// TIA Portal V18 export
FUNCTION_BLOCK "V90_Servo"   // FB2500, LAD
{ S7_Optimized_Access := 'TRUE' }
// stored: AutoNumber false, MemoryReserve 100, SetENOAutomatically false
   VAR
      Servo_380A1 { S7_SetPoint := 'True'} : "fbV90Ctrl";   // *
      Servo_381A1 { S7_SetPoint := 'True'} : "fbV90Ctrl";   // *
      Servo_382A1 { S7_SetPoint := 'True'} : "fbV90Ctrl";   // *
      Servo_383A1 { S7_SetPoint := 'True'} : "fbV90Ctrl";   // *
      Servo1 { S7_SetPoint := 'True'} : "SevroStart&PosCheck";
      Servo2 { S7_SetPoint := 'True'} : "SevroStart&PosCheck";
      Servo3 { S7_SetPoint := 'True'} : "SevroStart&PosCheck";
      Servo4 { S7_SetPoint := 'True'} : "SevroStart&PosCheck";
      Servo2SafetyPos { S7_SetPoint := 'True'} : DInt;
      Servo4SafetyPos { S7_SetPoint := 'True'} : DInt;
      IEC_Timer_0_Instance { S7_SetPoint := 'True'} : TON_TIME;
      P { S7_SetPoint := 'True'} : Array[0..10] of Bool;
      MC_MOVEJOG_Instance { S7_SetPoint := 'True'} : MC_MOVEJOG;
      MC_POWER_Instance { S7_SetPoint := 'True'} : MC_POWER;
      BasicPosControl { S7_SetPoint := 'True'} : BasicPosControl;
   END_VAR
   VAR_TEMP
      Sevro1ActPos : Real;
      Sevro1StartList : Bool;
      Sevro2ActPos : Real;
      Sevro2StartList : Bool;
      Sevro3ActPos : Real;
      Sevro3StartList : Bool;
      Sevro4ActPos : Real;
      Sevro4StartList : Bool;
      dummy : Bool;
      gotopos : Real;
      speed : Int;
   END_VAR
   VAR_TEMP   // added for the SCL form of the ladder/FBD networks
      _w1 : Bool;
      _w2 : Bool;
      _w3 : Bool;
      _w4 : Bool;
      _w5 : Bool;
   END_VAR
BEGIN

REGION Network 1: <<<<<<<<<<<<<<<<<<<<<380A1 Servo>>>>>>>>>>>>>>>>>>>>>>>>>
END_REGION

REGION Network 2: negtive motion/action/...automaticly
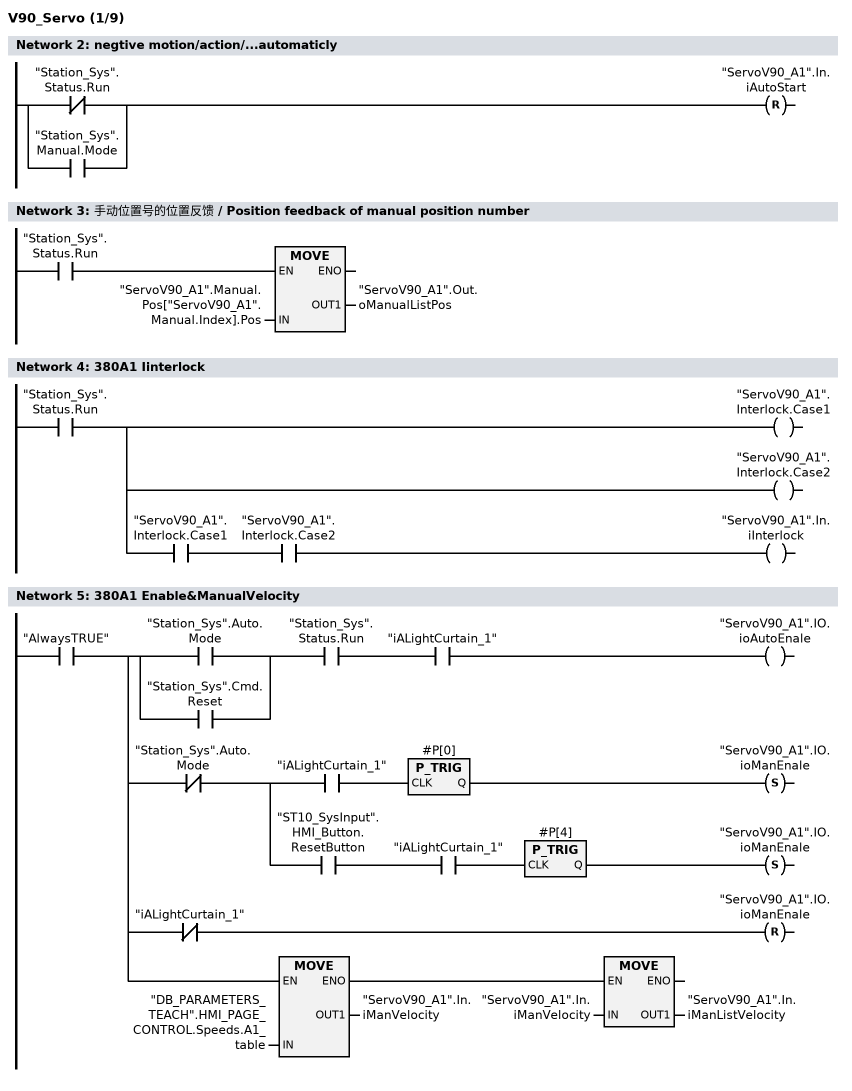
   RUNG wire#powerrail
      I_Contact( "Station_Sys".Status.Run )
      wire#w1
      R_Coil( "ServoV90_A1".In.iAutoStart )
   END_RUNG
   RUNG wire#powerrail
      Contact( "Station_Sys".Manual.Mode )
   END_RUNG wire#w1
   // the same network as SCL:
   IF NOT "Station_Sys".Status.Run OR "Station_Sys".Manual.Mode THEN
       "ServoV90_A1".In.iAutoStart := FALSE;
   END_IF;
END_REGION

REGION Network 3: 手动位置号的位置反馈 / Position feedback of manual position number
   RUNG wire#powerrail
      Contact( "Station_Sys".Status.Run )
      Move(in := "ServoV90_A1".Manual.Pos["ServoV90_A1".Manual.Index].Pos, out1 => "ServoV90_A1".Out.oManualListPos)
   END_RUNG
   // the same network as SCL:
   IF "Station_Sys".Status.Run THEN
       "ServoV90_A1".Out.oManualListPos := "ServoV90_A1".Manual.Pos["ServoV90_A1".Manual.Index].Pos;
   END_IF;
END_REGION

REGION Network 4: 380A1 Iinterlock
   RUNG wire#powerrail
      Contact( "Station_Sys".Status.Run )
      wire#w1
      Coil( "ServoV90_A1".Interlock.Case1 )
   END_RUNG
   RUNG wire#w1
      Coil( "ServoV90_A1".Interlock.Case2 )
   END_RUNG
   RUNG wire#w1
      Contact( "ServoV90_A1".Interlock.Case1 )
      Contact( "ServoV90_A1".Interlock.Case2 )
      Coil( "ServoV90_A1".In.iInterlock )
   END_RUNG
   // the same network as SCL:
   "ServoV90_A1".Interlock.Case1 := "Station_Sys".Status.Run;
   "ServoV90_A1".Interlock.Case2 := "Station_Sys".Status.Run;
   "ServoV90_A1".In.iInterlock := "Station_Sys".Status.Run AND "ServoV90_A1".Interlock.Case1 AND "ServoV90_A1".Interlock.Case2;
END_REGION

REGION Network 5: 380A1 Enable&ManualVelocity
   RUNG wire#powerrail
      Contact( "AlwaysTRUE" )
      wire#w1
      Contact( "Station_Sys".Auto.Mode )
      wire#w2
      Contact( "Station_Sys".Status.Run )
      Contact( "iALightCurtain_1" )
      Coil( "ServoV90_A1".IO.ioAutoEnale )
   END_RUNG
   RUNG wire#w1
      Contact( "Station_Sys".Cmd.Reset )
   END_RUNG wire#w2
   RUNG wire#w1
      I_Contact( "Station_Sys".Auto.Mode )
      wire#w3
      Contact( "iALightCurtain_1" )
      P_Trig( #P[0] )
      S_Coil( "ServoV90_A1".IO.ioManEnale )
   END_RUNG
   RUNG wire#w3
      Contact( "ST10_SysInput".HMI_Button.ResetButton )
      Contact( "iALightCurtain_1" )
      P_Trig( #P[4] )
      S_Coil( "ServoV90_A1".IO.ioManEnale )
   END_RUNG
   RUNG wire#w1
      I_Contact( "iALightCurtain_1" )
      R_Coil( "ServoV90_A1".IO.ioManEnale )
   END_RUNG
   RUNG wire#w1
      Move(in := "DB_PARAMETERS_TEACH".HMI_PAGE_CONTROL.Speeds.A1_table, out1 => "ServoV90_A1".In.iManVelocity)
      Move(in := "ServoV90_A1".In.iManVelocity, out1 => "ServoV90_A1".In.iManListVelocity)
   END_RUNG
   // the same network as SCL:
   "ServoV90_A1".IO.ioAutoEnale := "AlwaysTRUE" AND ("Station_Sys".Auto.Mode OR "Station_Sys".Cmd.Reset) AND "Station_Sys".Status.Run AND "iALightCurtain_1";
   #_w1 := "AlwaysTRUE" AND NOT "Station_Sys".Auto.Mode;
   #_w2 := #_w1 AND "iALightCurtain_1";
   #_w3 := #_w2 AND NOT #P[0];   // rising edge
   #P[0] := #_w2;
   IF #_w3 THEN "ServoV90_A1".IO.ioManEnale := TRUE; END_IF;
   #_w4 := #_w1 AND "ST10_SysInput".HMI_Button.ResetButton AND "iALightCurtain_1";
   #_w5 := #_w4 AND NOT #P[4];   // rising edge
   #P[4] := #_w4;
   IF #_w5 THEN "ServoV90_A1".IO.ioManEnale := TRUE; END_IF;
   IF "AlwaysTRUE" AND NOT "iALightCurtain_1" THEN "ServoV90_A1".IO.ioManEnale := FALSE; END_IF;
   IF "AlwaysTRUE" THEN
       "ServoV90_A1".In.iManVelocity := "DB_PARAMETERS_TEACH".HMI_PAGE_CONTROL.Speeds.A1_table;
       "ServoV90_A1".In.iManListVelocity := "ServoV90_A1".In.iManVelocity;
   END_IF;
END_REGION

REGION Network 6 (SCL): 380A1 RecipePosition
    IF "Station_Sys".Status.Run THEN
        "ServoV90_A1".Manual.Pos[1].Pos := "ServoV90_A1".Auto.Pos[1].Pos :=REAL_TO_DINT("Parameter".AxisRun.Axis[1].Pos1.Position*1000);
        "ServoV90_A1".Manual.Pos[1].Vel := "ServoV90_A1".Auto.Pos[1].Vel := "Parameter".AxisRun.Axis[1].Pos1.Speed;

        "ServoV90_A1".Manual.Pos[2].Pos := "ServoV90_A1".Auto.Pos[2].Pos := REAL_TO_DINT("Parameter".AxisRun.Axis[1].Pos2.Position*1000);
       "ServoV90_A1".Manual.Pos[2].Vel := "ServoV90_A1".Auto.Pos[2].Vel := "Parameter".AxisRun.Axis[1].Pos2.Speed;

       "ServoV90_A1".Manual.Pos[3].Pos := "ServoV90_A1".Auto.Pos[3].Pos := REAL_TO_DINT("Parameter".AxisRun.Axis[1].Pos3.Position*1000);
       "ServoV90_A1".Manual.Pos[3].Vel := "ServoV90_A1".Auto.Pos[3].Vel := "Parameter".AxisRun.Axis[1].Pos3.Speed;

       "ServoV90_A1".Manual.Pos[4].Pos := "ServoV90_A1".Auto.Pos[4].Pos := REAL_TO_DINT("Parameter".AxisRun.Axis[1].Pos4.Position*1000);
       "ServoV90_A1".Manual.Pos[4].Vel := "ServoV90_A1".Auto.Pos[4].Vel := "Parameter".AxisRun.Axis[1].Pos4.Speed;

       "ServoV90_A1".Manual.Pos[5].Pos := "ServoV90_A1".Auto.Pos[5].Pos := REAL_TO_DINT("Parameter".AxisRun.Axis[1].Pos5.Position*1000);
       "ServoV90_A1".Manual.Pos[5].Vel := "ServoV90_A1".Auto.Pos[5].Vel := "Parameter".AxisRun.Axis[1].Pos5.Speed;

       "ServoV90_A1".Manual.Pos[6].Pos := "ServoV90_A1".Auto.Pos[6].Pos := REAL_TO_DINT("Parameter".AxisRun.Axis[1].Pos6.Position*1000);
       "ServoV90_A1".Manual.Pos[6].Vel := "ServoV90_A1".Auto.Pos[6].Vel := "Parameter".AxisRun.Axis[1].Pos6.Speed;

       "ServoV90_A1".Manual.Pos[7].Pos := "ServoV90_A1".Auto.Pos[7].Pos := REAL_TO_DINT("Parameter".AxisRun.Axis[1].Pos7.Position*1000);
       "ServoV90_A1".Manual.Pos[7].Vel := "ServoV90_A1".Auto.Pos[7].Vel := "Parameter".AxisRun.Axis[1].Pos7.Speed;

       "ServoV90_A1".Manual.Pos[8].Pos := "ServoV90_A1".Auto.Pos[8].Pos := REAL_TO_DINT("Parameter".AxisRun.Axis[1].Pos8.Position*1000);
       "ServoV90_A1".Manual.Pos[8].Vel := "ServoV90_A1".Auto.Pos[8].Vel := "Parameter".AxisRun.Axis[1].Pos8.Speed;

       "ServoV90_A1".Manual.Pos[9].Pos := "ServoV90_A1".Auto.Pos[9].Pos := REAL_TO_DINT("Parameter".AxisRun.Axis[1].Pos9.Position*1000);
       "ServoV90_A1".Manual.Pos[9].Vel := "ServoV90_A1".Auto.Pos[9].Vel := "Parameter".AxisRun.Axis[1].Pos9.Speed;

   END_IF;
END_REGION

REGION Network 7: 380A1 FB
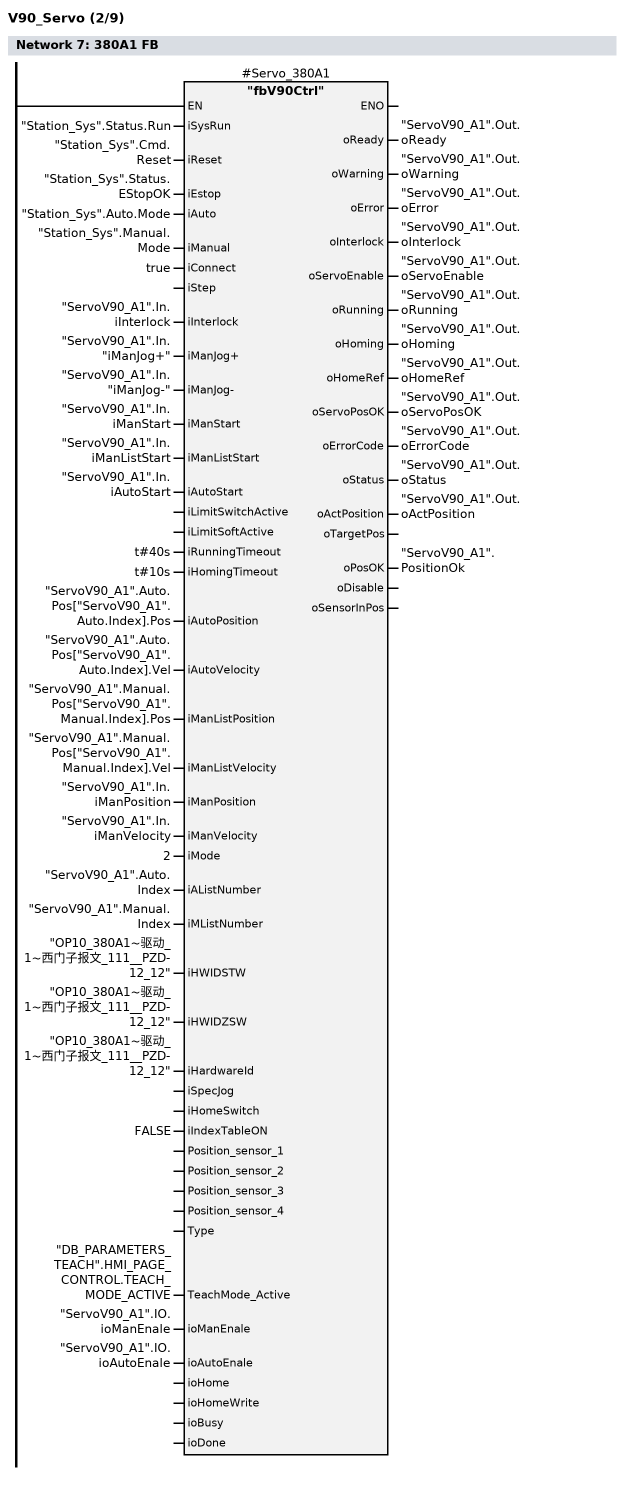
   RUNG wire#powerrail
      #Servo_380A1(iSysRun := "Station_Sys".Status.Run, iReset := "Station_Sys".Cmd.Reset, iEstop := "Station_Sys".Status.EStopOK, iAuto := "Station_Sys".Auto.Mode, iManual := "Station_Sys".Manual.Mode, iConnect := true, iStep :=, iInterlock := "ServoV90_A1".In.iInterlock, "iManJog+" := "ServoV90_A1".In."iManJog+", "iManJog-" := "ServoV90_A1".In."iManJog-", iManStart := "ServoV90_A1".In.iManStart, iManListStart := "ServoV90_A1".In.iManListStart, iAutoStart := "ServoV90_A1".In.iAutoStart, iLimitSwitchActive :=, iLimitSoftActive :=, iRunningTimeout := t#40s, iHomingTimeout := t#10s, iAutoPosition := "ServoV90_A1".Auto.Pos["ServoV90_A1".Auto.Index].Pos, iAutoVelocity := "ServoV90_A1".Auto.Pos["ServoV90_A1".Auto.Index].Vel, iManListPosition := "ServoV90_A1".Manual.Pos["ServoV90_A1".Manual.Index].Pos, iManListVelocity := "ServoV90_A1".Manual.Pos["ServoV90_A1".Manual.Index].Vel, iManPosition := "ServoV90_A1".In.iManPosition, iManVelocity := "ServoV90_A1".In.iManVelocity, iMode := 2, iAListNumber := "ServoV90_A1".Auto.Index, iMListNumber := "ServoV90_A1".Manual.Index, iHWIDSTW := "OP10_380A1~驱动_1~西门子报文_111__PZD-12_12", iHWIDZSW := "OP10_380A1~驱动_1~西门子报文_111__PZD-12_12", iHardwareId := "OP10_380A1~驱动_1~西门子报文_111__PZD-12_12", iSpecJog :=, iHomeSwitch :=, iIndexTableON := FALSE, Position_sensor_1 :=, Position_sensor_2 :=, Position_sensor_3 :=, Position_sensor_4 :=, "Type" :=, TeachMode_Active := "DB_PARAMETERS_TEACH".HMI_PAGE_CONTROL.TEACH_MODE_ACTIVE, ioManEnale := "ServoV90_A1".IO.ioManEnale, ioAutoEnale := "ServoV90_A1".IO.ioAutoEnale, ioHome :=, ioHomeWrite :=, ioBusy :=, ioDone :=, oReady => "ServoV90_A1".Out.oReady, oWarning => "ServoV90_A1".Out.oWarning, oError => "ServoV90_A1".Out.oError, oInterlock => "ServoV90_A1".Out.oInterlock, oServoEnable => "ServoV90_A1".Out.oServoEnable, oRunning => "ServoV90_A1".Out.oRunning, oHoming => "ServoV90_A1".Out.oHoming, oHomeRef => "ServoV90_A1".Out.oHomeRef, oServoPosOK => "ServoV90_A1".Out.oServoPosOK, oErrorCode => "ServoV90_A1".Out.oErrorCode, oStatus => "ServoV90_A1".Out.oStatus, oActPosition => "ServoV90_A1".Out.oActPosition, oTargetPos =>, oPosOK => "ServoV90_A1".PositionOk, oDisable =>, oSensorInPos =>)
   END_RUNG
   // the same network as SCL:
   #Servo_380A1(iSysRun := "Station_Sys".Status.Run,   // "fbV90Ctrl"
                iReset := "Station_Sys".Cmd.Reset,
                iEstop := "Station_Sys".Status.EStopOK,
                iAuto := "Station_Sys".Auto.Mode,
                iManual := "Station_Sys".Manual.Mode,
                iConnect := true,
                iInterlock := "ServoV90_A1".In.iInterlock,
                "iManJog+" := "ServoV90_A1".In."iManJog+",
                "iManJog-" := "ServoV90_A1".In."iManJog-",
                iManStart := "ServoV90_A1".In.iManStart,
                iManListStart := "ServoV90_A1".In.iManListStart,
                iAutoStart := "ServoV90_A1".In.iAutoStart,
                iRunningTimeout := t#40s,
                iHomingTimeout := t#10s,
                iAutoPosition := "ServoV90_A1".Auto.Pos["ServoV90_A1".Auto.Index].Pos,
                iAutoVelocity := "ServoV90_A1".Auto.Pos["ServoV90_A1".Auto.Index].Vel,
                iManListPosition := "ServoV90_A1".Manual.Pos["ServoV90_A1".Manual.Index].Pos,
                iManListVelocity := "ServoV90_A1".Manual.Pos["ServoV90_A1".Manual.Index].Vel,
                iManPosition := "ServoV90_A1".In.iManPosition,
                iManVelocity := "ServoV90_A1".In.iManVelocity,
                iMode := 2,
                iAListNumber := "ServoV90_A1".Auto.Index,
                iMListNumber := "ServoV90_A1".Manual.Index,
                iHWIDSTW := "OP10_380A1~驱动_1~西门子报文_111__PZD-12_12",
                iHWIDZSW := "OP10_380A1~驱动_1~西门子报文_111__PZD-12_12",
                iHardwareId := "OP10_380A1~驱动_1~西门子报文_111__PZD-12_12",
                iIndexTableON := FALSE,
                TeachMode_Active := "DB_PARAMETERS_TEACH".HMI_PAGE_CONTROL.TEACH_MODE_ACTIVE,
                ioManEnale := "ServoV90_A1".IO.ioManEnale,
                ioAutoEnale := "ServoV90_A1".IO.ioAutoEnale,
                oReady => "ServoV90_A1".Out.oReady,
                oWarning => "ServoV90_A1".Out.oWarning,
                oError => "ServoV90_A1".Out.oError,
                oInterlock => "ServoV90_A1".Out.oInterlock,
                oServoEnable => "ServoV90_A1".Out.oServoEnable,
                oRunning => "ServoV90_A1".Out.oRunning,
                oHoming => "ServoV90_A1".Out.oHoming,
                oHomeRef => "ServoV90_A1".Out.oHomeRef,
                oServoPosOK => "ServoV90_A1".Out.oServoPosOK,
                oErrorCode => "ServoV90_A1".Out.oErrorCode,
                oStatus => "ServoV90_A1".Out.oStatus,
                oActPosition => "ServoV90_A1".Out.oActPosition,
                oPosOK => "ServoV90_A1".PositionOk);
END_REGION

REGION Network 8 (SCL): 故障显示 / Fault indication
   //"ST70_DeviceError".Servo1.ServoDriverError := "ServoV90_A1".Out.oError;
END_REGION

REGION Network 9: <<<<<<<<<<<<<<<<<<<<<381A1 Servo>>>>>>>>>>>>>>>>>>>>>>>>>
END_REGION

REGION Network 10: negtive motion/action/...automaticly
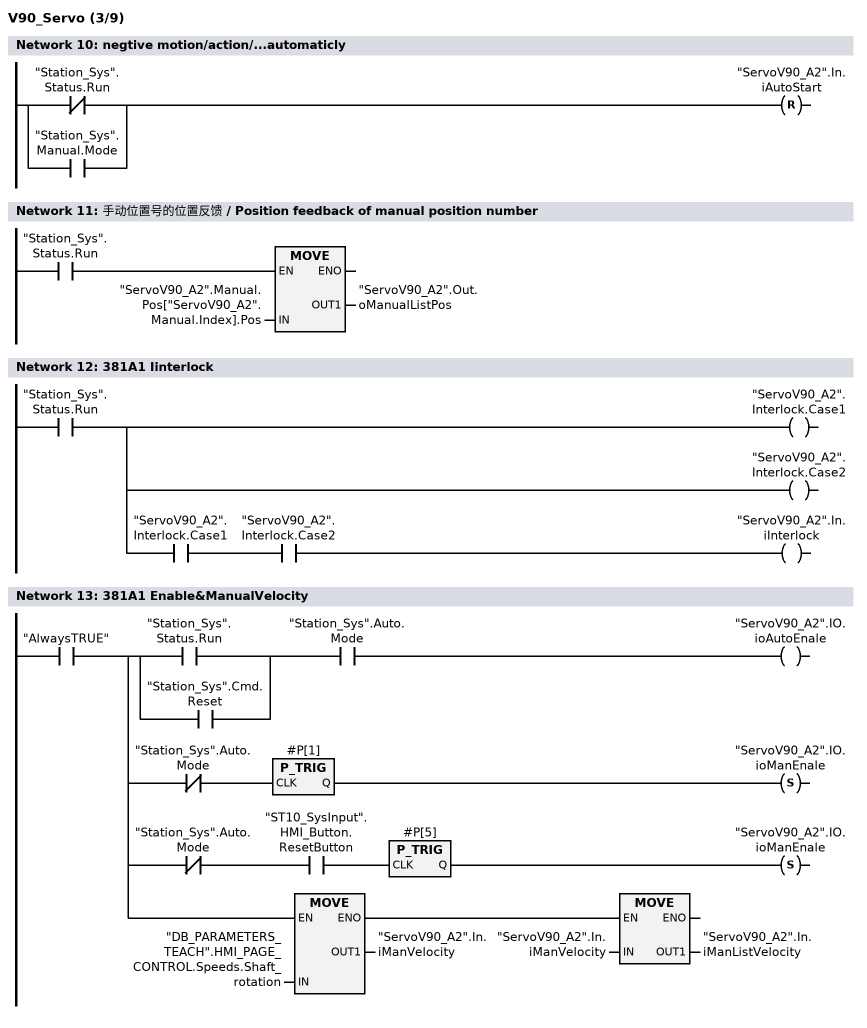
   RUNG wire#powerrail
      I_Contact( "Station_Sys".Status.Run )
      wire#w1
      R_Coil( "ServoV90_A2".In.iAutoStart )
   END_RUNG
   RUNG wire#powerrail
      Contact( "Station_Sys".Manual.Mode )
   END_RUNG wire#w1
   // the same network as SCL:
   IF NOT "Station_Sys".Status.Run OR "Station_Sys".Manual.Mode THEN
       "ServoV90_A2".In.iAutoStart := FALSE;
   END_IF;
END_REGION

REGION Network 11: 手动位置号的位置反馈 / Position feedback of manual position number
   RUNG wire#powerrail
      Contact( "Station_Sys".Status.Run )
      Move(in := "ServoV90_A2".Manual.Pos["ServoV90_A2".Manual.Index].Pos, out1 => "ServoV90_A2".Out.oManualListPos)
   END_RUNG
   // the same network as SCL:
   IF "Station_Sys".Status.Run THEN
       "ServoV90_A2".Out.oManualListPos := "ServoV90_A2".Manual.Pos["ServoV90_A2".Manual.Index].Pos;
   END_IF;
END_REGION

REGION Network 12: 381A1 Iinterlock
   RUNG wire#powerrail
      Contact( "Station_Sys".Status.Run )
      wire#w1
      Coil( "ServoV90_A2".Interlock.Case1 )
   END_RUNG
   RUNG wire#w1
      Coil( "ServoV90_A2".Interlock.Case2 )
   END_RUNG
   RUNG wire#w1
      Contact( "ServoV90_A2".Interlock.Case1 )
      Contact( "ServoV90_A2".Interlock.Case2 )
      Coil( "ServoV90_A2".In.iInterlock )
   END_RUNG
   // the same network as SCL:
   "ServoV90_A2".Interlock.Case1 := "Station_Sys".Status.Run;
   "ServoV90_A2".Interlock.Case2 := "Station_Sys".Status.Run;
   "ServoV90_A2".In.iInterlock := "Station_Sys".Status.Run AND "ServoV90_A2".Interlock.Case1 AND "ServoV90_A2".Interlock.Case2;
END_REGION

REGION Network 13: 381A1 Enable&ManualVelocity
   RUNG wire#powerrail
      Contact( "AlwaysTRUE" )
      wire#w1
      Contact( "Station_Sys".Status.Run )
      wire#w2
      Contact( "Station_Sys".Auto.Mode )
      Coil( "ServoV90_A2".IO.ioAutoEnale )
   END_RUNG
   RUNG wire#w1
      Contact( "Station_Sys".Cmd.Reset )
   END_RUNG wire#w2
   RUNG wire#w1
      I_Contact( "Station_Sys".Auto.Mode )
      P_Trig( #P[1] )
      S_Coil( "ServoV90_A2".IO.ioManEnale )
   END_RUNG
   RUNG wire#w1
      I_Contact( "Station_Sys".Auto.Mode )
      Contact( "ST10_SysInput".HMI_Button.ResetButton )
      P_Trig( #P[5] )
      S_Coil( "ServoV90_A2".IO.ioManEnale )
   END_RUNG
   RUNG wire#w1
      Move(in := "DB_PARAMETERS_TEACH".HMI_PAGE_CONTROL.Speeds.Shaft_rotation, out1 => "ServoV90_A2".In.iManVelocity)
      Move(in := "ServoV90_A2".In.iManVelocity, out1 => "ServoV90_A2".In.iManListVelocity)
   END_RUNG
   // the same network as SCL:
   "ServoV90_A2".IO.ioAutoEnale := "AlwaysTRUE" AND ("Station_Sys".Status.Run OR "Station_Sys".Cmd.Reset) AND "Station_Sys".Auto.Mode;
   #_w1 := "AlwaysTRUE" AND NOT "Station_Sys".Auto.Mode;
   #_w2 := #_w1 AND NOT #P[1];   // rising edge
   #P[1] := #_w1;
   IF #_w2 THEN "ServoV90_A2".IO.ioManEnale := TRUE; END_IF;
   #_w3 := "AlwaysTRUE" AND NOT "Station_Sys".Auto.Mode AND "ST10_SysInput".HMI_Button.ResetButton;
   #_w4 := #_w3 AND NOT #P[5];   // rising edge
   #P[5] := #_w3;
   IF #_w4 THEN "ServoV90_A2".IO.ioManEnale := TRUE; END_IF;
   IF "AlwaysTRUE" THEN
       "ServoV90_A2".In.iManVelocity := "DB_PARAMETERS_TEACH".HMI_PAGE_CONTROL.Speeds.Shaft_rotation;
       "ServoV90_A2".In.iManListVelocity := "ServoV90_A2".In.iManVelocity;
   END_IF;
END_REGION

REGION Network 14 (SCL): 381A1 RecipePosition
    IF "Station_Sys".Status.Run THEN
        "ServoV90_A2".Manual.Pos[1].Pos := "ServoV90_A2".Auto.Pos[1].Pos := REAL_TO_DINT("Parameter".AxisRun.Axis[2].Pos1.Position*1000);
       "ServoV90_A2".Manual.Pos[1].Vel := "ServoV90_A2".Auto.Pos[1].Vel := "Parameter".AxisRun.Axis[2].Pos1.Speed;

       "ServoV90_A2".Manual.Pos[2].Pos := "ServoV90_A2".Auto.Pos[2].Pos := REAL_TO_DINT("Parameter".AxisRun.Axis[2].Pos2.Position*1000);
       "ServoV90_A2".Manual.Pos[2].Vel := "ServoV90_A2".Auto.Pos[2].Vel := "Parameter".AxisRun.Axis[2].Pos2.Speed;

       "ServoV90_A2".Manual.Pos[3].Pos := "ServoV90_A2".Auto.Pos[3].Pos := REAL_TO_DINT("Parameter".AxisRun.Axis[2].Pos3.Position*1000);
       "ServoV90_A2".Manual.Pos[3].Vel := "ServoV90_A2".Auto.Pos[3].Vel := "Parameter".AxisRun.Axis[2].Pos3.Speed;

       "ServoV90_A2".Manual.Pos[4].Pos := "ServoV90_A2".Auto.Pos[4].Pos := REAL_TO_DINT("Parameter".AxisRun.Axis[2].Pos4.Position*1000);
       "ServoV90_A2".Manual.Pos[4].Vel := "ServoV90_A2".Auto.Pos[4].Vel := "Parameter".AxisRun.Axis[2].Pos4.Speed;

       "ServoV90_A2".Manual.Pos[5].Pos := "ServoV90_A2".Auto.Pos[5].Pos := REAL_TO_DINT("Parameter".AxisRun.Axis[2].Pos5.Position*1000);
       "ServoV90_A2".Manual.Pos[5].Vel := "ServoV90_A2".Auto.Pos[5].Vel := "Parameter".AxisRun.Axis[2].Pos5.Speed;

       "ServoV90_A2".Manual.Pos[6].Pos := "ServoV90_A2".Auto.Pos[6].Pos := REAL_TO_DINT("Parameter".AxisRun.Axis[2].Pos6.Position*1000);
       "ServoV90_A2".Manual.Pos[6].Vel := "ServoV90_A2".Auto.Pos[6].Vel := "Parameter".AxisRun.Axis[2].Pos6.Speed;

       "ServoV90_A2".Manual.Pos[7].Pos := "ServoV90_A2".Auto.Pos[7].Pos := REAL_TO_DINT("Parameter".AxisRun.Axis[2].Pos7.Position*1000);
       "ServoV90_A2".Manual.Pos[7].Vel := "ServoV90_A2".Auto.Pos[7].Vel := "Parameter".AxisRun.Axis[2].Pos7.Speed;

       "ServoV90_A2".Manual.Pos[8].Pos := "ServoV90_A2".Auto.Pos[8].Pos := REAL_TO_DINT("Parameter".AxisRun.Axis[2].Pos8.Position*1000);
       "ServoV90_A2".Manual.Pos[8].Vel := "ServoV90_A2".Auto.Pos[8].Vel := "Parameter".AxisRun.Axis[2].Pos8.Speed;

       "ServoV90_A2".Manual.Pos[9].Pos := "ServoV90_A2".Auto.Pos[9].Pos := REAL_TO_DINT("Parameter".AxisRun.Axis[2].Pos9.Position*1000);
       "ServoV90_A2".Manual.Pos[9].Vel := "ServoV90_A2".Auto.Pos[9].Vel := "Parameter".AxisRun.Axis[2].Pos9.Speed;

       "ServoV90_A2".Manual.Pos[10].Pos := "ServoV90_A2".Auto.Pos[10].Pos := REAL_TO_DINT("Parameter".AxisRun.Axis[2].Pos10.Position*1000);
       "ServoV90_A2".Manual.Pos[10].Vel := "ServoV90_A2".Auto.Pos[10].Vel := "Parameter".AxisRun.Axis[2].Pos10.Speed;
   END_IF;
END_REGION

REGION Network 15: 381A1 FB
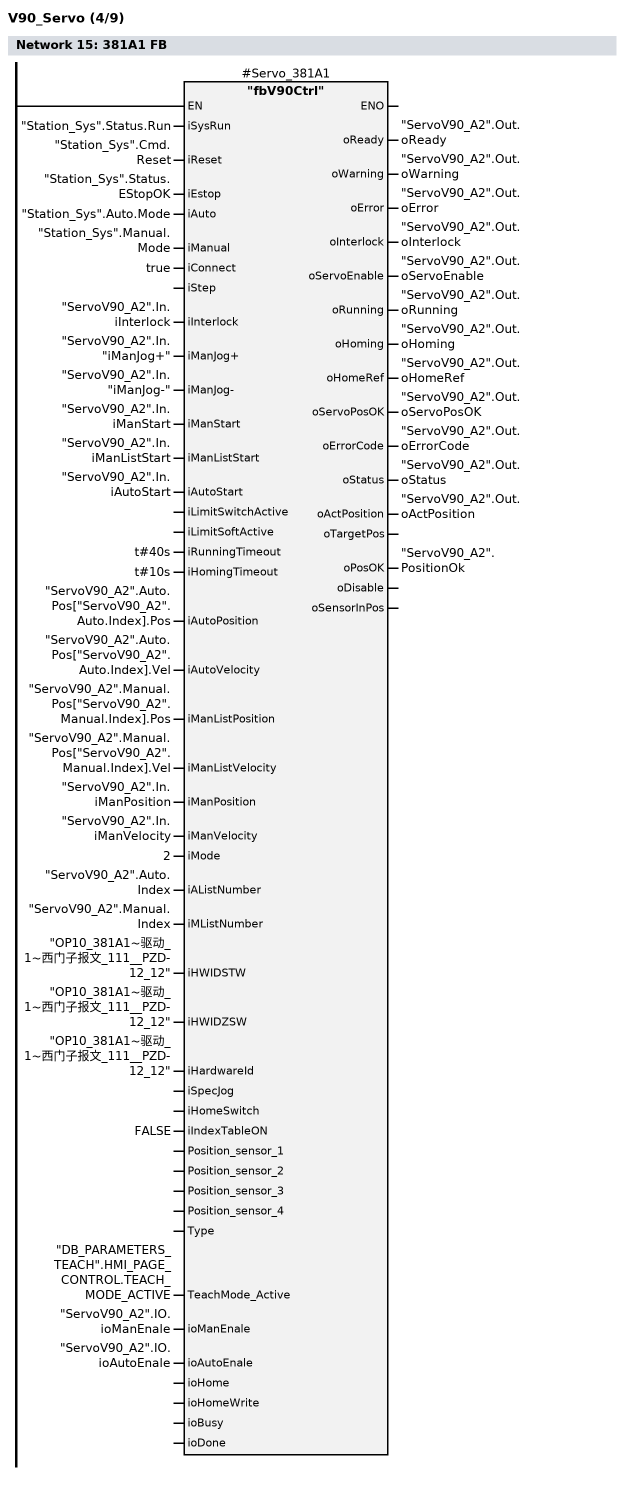
   RUNG wire#powerrail
      #Servo_381A1(iSysRun := "Station_Sys".Status.Run, iReset := "Station_Sys".Cmd.Reset, iEstop := "Station_Sys".Status.EStopOK, iAuto := "Station_Sys".Auto.Mode, iManual := "Station_Sys".Manual.Mode, iConnect := true, iStep :=, iInterlock := "ServoV90_A2".In.iInterlock, "iManJog+" := "ServoV90_A2".In."iManJog+", "iManJog-" := "ServoV90_A2".In."iManJog-", iManStart := "ServoV90_A2".In.iManStart, iManListStart := "ServoV90_A2".In.iManListStart, iAutoStart := "ServoV90_A2".In.iAutoStart, iLimitSwitchActive :=, iLimitSoftActive :=, iRunningTimeout := t#40s, iHomingTimeout := t#10s, iAutoPosition := "ServoV90_A2".Auto.Pos["ServoV90_A2".Auto.Index].Pos, iAutoVelocity := "ServoV90_A2".Auto.Pos["ServoV90_A2".Auto.Index].Vel, iManListPosition := "ServoV90_A2".Manual.Pos["ServoV90_A2".Manual.Index].Pos, iManListVelocity := "ServoV90_A2".Manual.Pos["ServoV90_A2".Manual.Index].Vel, iManPosition := "ServoV90_A2".In.iManPosition, iManVelocity := "ServoV90_A2".In.iManVelocity, iMode := 2, iAListNumber := "ServoV90_A2".Auto.Index, iMListNumber := "ServoV90_A2".Manual.Index, iHWIDSTW := "OP10_381A1~驱动_1~西门子报文_111__PZD-12_12", iHWIDZSW := "OP10_381A1~驱动_1~西门子报文_111__PZD-12_12", iHardwareId := "OP10_381A1~驱动_1~西门子报文_111__PZD-12_12", iSpecJog :=, iHomeSwitch :=, iIndexTableON := FALSE, Position_sensor_1 :=, Position_sensor_2 :=, Position_sensor_3 :=, Position_sensor_4 :=, "Type" :=, TeachMode_Active := "DB_PARAMETERS_TEACH".HMI_PAGE_CONTROL.TEACH_MODE_ACTIVE, ioManEnale := "ServoV90_A2".IO.ioManEnale, ioAutoEnale := "ServoV90_A2".IO.ioAutoEnale, ioHome :=, ioHomeWrite :=, ioBusy :=, ioDone :=, oReady => "ServoV90_A2".Out.oReady, oWarning => "ServoV90_A2".Out.oWarning, oError => "ServoV90_A2".Out.oError, oInterlock => "ServoV90_A2".Out.oInterlock, oServoEnable => "ServoV90_A2".Out.oServoEnable, oRunning => "ServoV90_A2".Out.oRunning, oHoming => "ServoV90_A2".Out.oHoming, oHomeRef => "ServoV90_A2".Out.oHomeRef, oServoPosOK => "ServoV90_A2".Out.oServoPosOK, oErrorCode => "ServoV90_A2".Out.oErrorCode, oStatus => "ServoV90_A2".Out.oStatus, oActPosition => "ServoV90_A2".Out.oActPosition, oTargetPos =>, oPosOK => "ServoV90_A2".PositionOk, oDisable =>, oSensorInPos =>)
   END_RUNG
   // the same network as SCL:
   #Servo_381A1(iSysRun := "Station_Sys".Status.Run,   // "fbV90Ctrl"
                iReset := "Station_Sys".Cmd.Reset,
                iEstop := "Station_Sys".Status.EStopOK,
                iAuto := "Station_Sys".Auto.Mode,
                iManual := "Station_Sys".Manual.Mode,
                iConnect := true,
                iInterlock := "ServoV90_A2".In.iInterlock,
                "iManJog+" := "ServoV90_A2".In."iManJog+",
                "iManJog-" := "ServoV90_A2".In."iManJog-",
                iManStart := "ServoV90_A2".In.iManStart,
                iManListStart := "ServoV90_A2".In.iManListStart,
                iAutoStart := "ServoV90_A2".In.iAutoStart,
                iRunningTimeout := t#40s,
                iHomingTimeout := t#10s,
                iAutoPosition := "ServoV90_A2".Auto.Pos["ServoV90_A2".Auto.Index].Pos,
                iAutoVelocity := "ServoV90_A2".Auto.Pos["ServoV90_A2".Auto.Index].Vel,
                iManListPosition := "ServoV90_A2".Manual.Pos["ServoV90_A2".Manual.Index].Pos,
                iManListVelocity := "ServoV90_A2".Manual.Pos["ServoV90_A2".Manual.Index].Vel,
                iManPosition := "ServoV90_A2".In.iManPosition,
                iManVelocity := "ServoV90_A2".In.iManVelocity,
                iMode := 2,
                iAListNumber := "ServoV90_A2".Auto.Index,
                iMListNumber := "ServoV90_A2".Manual.Index,
                iHWIDSTW := "OP10_381A1~驱动_1~西门子报文_111__PZD-12_12",
                iHWIDZSW := "OP10_381A1~驱动_1~西门子报文_111__PZD-12_12",
                iHardwareId := "OP10_381A1~驱动_1~西门子报文_111__PZD-12_12",
                iIndexTableON := FALSE,
                TeachMode_Active := "DB_PARAMETERS_TEACH".HMI_PAGE_CONTROL.TEACH_MODE_ACTIVE,
                ioManEnale := "ServoV90_A2".IO.ioManEnale,
                ioAutoEnale := "ServoV90_A2".IO.ioAutoEnale,
                oReady => "ServoV90_A2".Out.oReady,
                oWarning => "ServoV90_A2".Out.oWarning,
                oError => "ServoV90_A2".Out.oError,
                oInterlock => "ServoV90_A2".Out.oInterlock,
                oServoEnable => "ServoV90_A2".Out.oServoEnable,
                oRunning => "ServoV90_A2".Out.oRunning,
                oHoming => "ServoV90_A2".Out.oHoming,
                oHomeRef => "ServoV90_A2".Out.oHomeRef,
                oServoPosOK => "ServoV90_A2".Out.oServoPosOK,
                oErrorCode => "ServoV90_A2".Out.oErrorCode,
                oStatus => "ServoV90_A2".Out.oStatus,
                oActPosition => "ServoV90_A2".Out.oActPosition,
                oPosOK => "ServoV90_A2".PositionOk);
END_REGION

REGION Network 16 (SCL): 故障显示 / Fault indication
   //"ST70_DeviceError".Servo2.ServoDriverError := "ServoV90_A2".Out.oError;
   //

   "ServoV90_A3".Auto.Index := "ServoV90_A3".Auto.Index;
END_REGION

REGION Network 17: <<<<<<<<<<<<<<<<<<<<<382A1 Servo>>>>>>>>>>>>>>>>>>>>>>>>>
END_REGION

REGION Network 18: <<<<<<<<<<<<<<<<<<<<<382A1 Servo>>>>>>>>>>>>>>>>>>>>>>>>> / $$$$####### NEW TECHNOLOGY OBJECTS #################
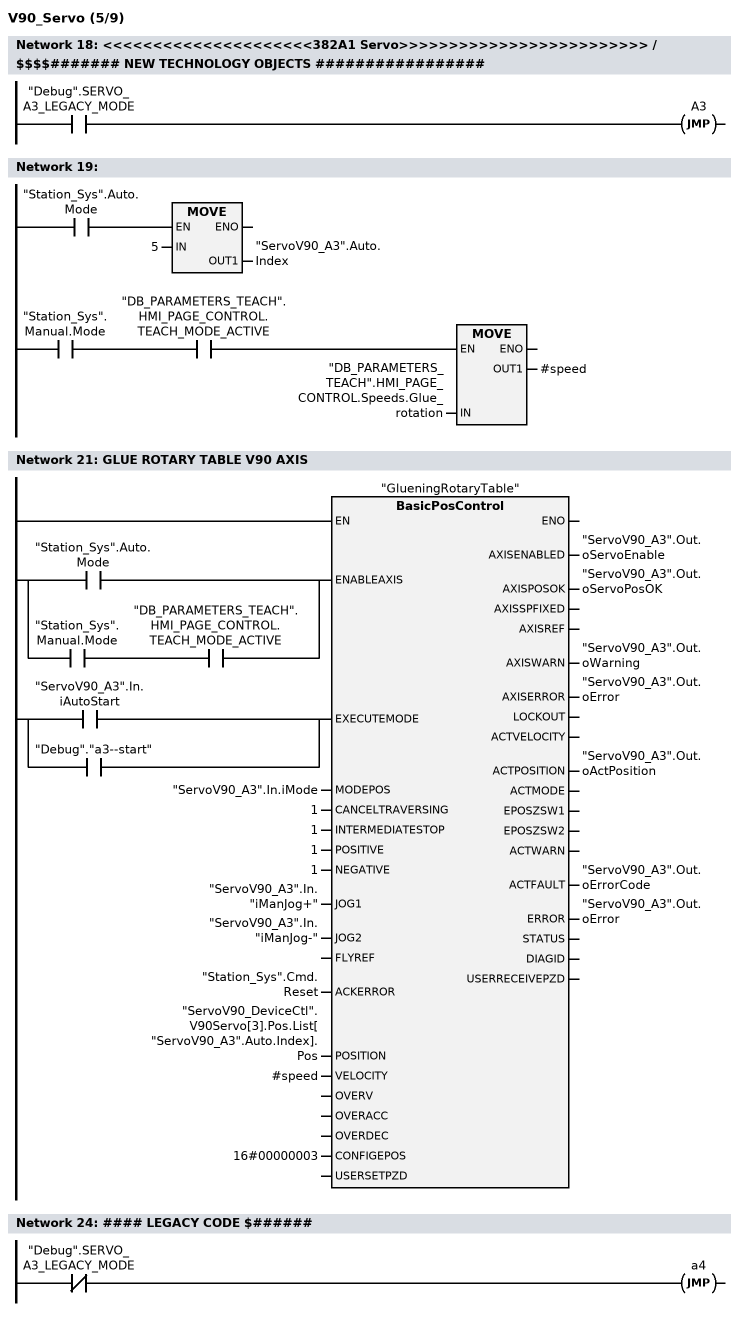
   RUNG wire#powerrail
      Contact( "Debug".SERVO_A3_LEGACY_MODE )
      JumpCoil( A3 )
   END_RUNG
   // the same network as SCL:
   IF "Debug".SERVO_A3_LEGACY_MODE THEN GOTO A3; END_IF;
END_REGION

REGION Network 19
   RUNG wire#powerrail
      Contact( "Station_Sys".Auto.Mode )
      Move(in := 5, out1 => "ServoV90_A3".Auto.Index)
   END_RUNG
   RUNG wire#powerrail
      Contact( "Station_Sys".Manual.Mode )
      Contact( "DB_PARAMETERS_TEACH".HMI_PAGE_CONTROL.TEACH_MODE_ACTIVE )
      Move(in := "DB_PARAMETERS_TEACH".HMI_PAGE_CONTROL.Speeds.Glue_rotation, out1 => #speed)
   END_RUNG
   // the same network as SCL:
   IF "Station_Sys".Auto.Mode THEN "ServoV90_A3".Auto.Index := 5; END_IF;
   IF "Station_Sys".Manual.Mode AND "DB_PARAMETERS_TEACH".HMI_PAGE_CONTROL.TEACH_MODE_ACTIVE THEN
       #speed := "DB_PARAMETERS_TEACH".HMI_PAGE_CONTROL.Speeds.Glue_rotation;
   END_IF;
END_REGION

REGION Network 21: GLUE ROTARY TABLE V90 AXIS
   RUNG wire#powerrail
      "GlueningRotaryTable".BasicPosControl(EnableAxis := wire#w1, ExecuteMode := wire#w2, ModePos := "ServoV90_A3".In.iMode, CancelTraversing := 1, IntermediateStop := 1, Positive := 1, Negative := 1, Jog1 := "ServoV90_A3".In."iManJog+", Jog2 := "ServoV90_A3".In."iManJog-", FlyRef :=, AckError := "Station_Sys".Cmd.Reset, Position := "ServoV90_DeviceCtl".V90Servo[3].Pos.List["ServoV90_A3".Auto.Index].Pos, Velocity := #speed, OverV :=, OverAcc :=, OverDec :=, ConfigEPos := 16#00000003, UserSetPZD :=, AxisEnabled => "ServoV90_A3".Out.oServoEnable, AxisPosOk => "ServoV90_A3".Out.oServoPosOK, AxisSpFixed =>, AxisRef =>, AxisWarn => "ServoV90_A3".Out.oWarning, AxisError => "ServoV90_A3".Out.oError, Lockout =>, ActVelocity =>, ActPosition => "ServoV90_A3".Out.oActPosition, ActMode =>, EPosZSW1 =>, EPosZSW2 =>, ActWarn =>, ActFault => "ServoV90_A3".Out.oErrorCode, Error => "ServoV90_A3".Out.oError, Status =>, DiagId =>, UserReceivePZD =>)
   END_RUNG
   RUNG wire#powerrail
      Contact( "Station_Sys".Auto.Mode )
   END_RUNG wire#w1
   RUNG wire#powerrail
      Contact( "Station_Sys".Manual.Mode )
      Contact( "DB_PARAMETERS_TEACH".HMI_PAGE_CONTROL.TEACH_MODE_ACTIVE )
   END_RUNG wire#w1
   RUNG wire#powerrail
      Contact( "ServoV90_A3".In.iAutoStart )
   END_RUNG wire#w2
   RUNG wire#powerrail
      Contact( "Debug"."a3--start" )
   END_RUNG wire#w2
   // the same network as SCL:
   "GlueningRotaryTable"(EnableAxis := "Station_Sys".Auto.Mode OR ("Station_Sys".Manual.Mode AND "DB_PARAMETERS_TEACH".HMI_PAGE_CONTROL.TEACH_MODE_ACTIVE),   // BasicPosControl
                         ExecuteMode := "ServoV90_A3".In.iAutoStart OR "Debug"."a3--start",
                         ModePos := "ServoV90_A3".In.iMode,
                         CancelTraversing := 1,
                         IntermediateStop := 1,
                         Positive := 1,
                         Negative := 1,
                         Jog1 := "ServoV90_A3".In."iManJog+",
                         Jog2 := "ServoV90_A3".In."iManJog-",
                         AckError := "Station_Sys".Cmd.Reset,
                         Position := "ServoV90_DeviceCtl".V90Servo[3].Pos.List["ServoV90_A3".Auto.Index].Pos,
                         Velocity := #speed,
                         ConfigEPos := 16#00000003,
                         AxisEnabled => "ServoV90_A3".Out.oServoEnable,
                         AxisPosOk => "ServoV90_A3".Out.oServoPosOK,
                         AxisWarn => "ServoV90_A3".Out.oWarning,
                         AxisError => "ServoV90_A3".Out.oError,
                         ActPosition => "ServoV90_A3".Out.oActPosition,
                         ActFault => "ServoV90_A3".Out.oErrorCode,
                         Error => "ServoV90_A3".Out.oError);
END_REGION

REGION Network 23: <<<<<<<<<<<<<<<<<<<<<382A1 Servo>>>>>>>>>>>>>>>>>>>>>>>>> / ################# ##################################
END_REGION

REGION Network 24: #### LEGACY CODE $######
   RUNG wire#powerrail
      I_Contact( "Debug".SERVO_A3_LEGACY_MODE )
      JumpCoil( a4 )
   END_RUNG
   // the same network as SCL:
   IF NOT "Debug".SERVO_A3_LEGACY_MODE THEN GOTO a4; END_IF;
END_REGION

REGION Network 25: negtive motion/action/...automaticly
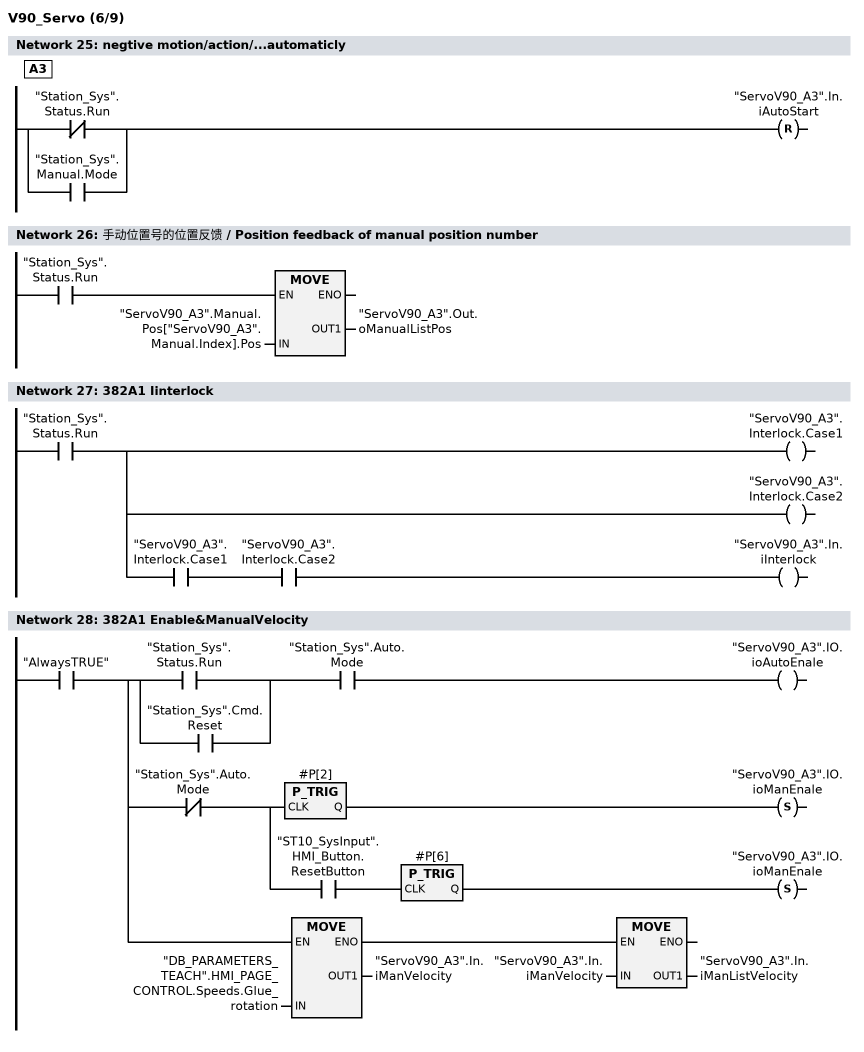
   Label( A3 )
   RUNG wire#powerrail
      I_Contact( "Station_Sys".Status.Run )
      wire#w1
      R_Coil( "ServoV90_A3".In.iAutoStart )
   END_RUNG
   RUNG wire#powerrail
      Contact( "Station_Sys".Manual.Mode )
   END_RUNG wire#w1
   // the same network as SCL:
   A3:
   IF NOT "Station_Sys".Status.Run OR "Station_Sys".Manual.Mode THEN
       "ServoV90_A3".In.iAutoStart := FALSE;
   END_IF;
END_REGION

REGION Network 26: 手动位置号的位置反馈 / Position feedback of manual position number
   RUNG wire#powerrail
      Contact( "Station_Sys".Status.Run )
      Move(in := "ServoV90_A3".Manual.Pos["ServoV90_A3".Manual.Index].Pos, out1 => "ServoV90_A3".Out.oManualListPos)
   END_RUNG
   // the same network as SCL:
   IF "Station_Sys".Status.Run THEN
       "ServoV90_A3".Out.oManualListPos := "ServoV90_A3".Manual.Pos["ServoV90_A3".Manual.Index].Pos;
   END_IF;
END_REGION

REGION Network 27: 382A1 Iinterlock
   RUNG wire#powerrail
      Contact( "Station_Sys".Status.Run )
      wire#w1
      Coil( "ServoV90_A3".Interlock.Case1 )
   END_RUNG
   RUNG wire#w1
      Coil( "ServoV90_A3".Interlock.Case2 )
   END_RUNG
   RUNG wire#w1
      Contact( "ServoV90_A3".Interlock.Case1 )
      Contact( "ServoV90_A3".Interlock.Case2 )
      Coil( "ServoV90_A3".In.iInterlock )
   END_RUNG
   // the same network as SCL:
   "ServoV90_A3".Interlock.Case1 := "Station_Sys".Status.Run;
   "ServoV90_A3".Interlock.Case2 := "Station_Sys".Status.Run;
   "ServoV90_A3".In.iInterlock := "Station_Sys".Status.Run AND "ServoV90_A3".Interlock.Case1 AND "ServoV90_A3".Interlock.Case2;
END_REGION

REGION Network 28: 382A1 Enable&ManualVelocity
   RUNG wire#powerrail
      Contact( "AlwaysTRUE" )
      wire#w1
      Contact( "Station_Sys".Status.Run )
      wire#w2
      Contact( "Station_Sys".Auto.Mode )
      Coil( "ServoV90_A3".IO.ioAutoEnale )
   END_RUNG
   RUNG wire#w1
      Contact( "Station_Sys".Cmd.Reset )
   END_RUNG wire#w2
   RUNG wire#w1
      I_Contact( "Station_Sys".Auto.Mode )
      wire#w3
      P_Trig( #P[2] )
      S_Coil( "ServoV90_A3".IO.ioManEnale )
   END_RUNG
   RUNG wire#w3
      Contact( "ST10_SysInput".HMI_Button.ResetButton )
      P_Trig( #P[6] )
      S_Coil( "ServoV90_A3".IO.ioManEnale )
   END_RUNG
   RUNG wire#w1
      Move(in := "DB_PARAMETERS_TEACH".HMI_PAGE_CONTROL.Speeds.Glue_rotation, out1 => "ServoV90_A3".In.iManVelocity)
      Move(in := "ServoV90_A3".In.iManVelocity, out1 => "ServoV90_A3".In.iManListVelocity)
   END_RUNG
   // the same network as SCL:
   "ServoV90_A3".IO.ioAutoEnale := "AlwaysTRUE" AND ("Station_Sys".Status.Run OR "Station_Sys".Cmd.Reset) AND "Station_Sys".Auto.Mode;
   #_w1 := "AlwaysTRUE" AND NOT "Station_Sys".Auto.Mode;
   #_w2 := #_w1 AND NOT #P[2];   // rising edge
   #P[2] := #_w1;
   IF #_w2 THEN "ServoV90_A3".IO.ioManEnale := TRUE; END_IF;
   #_w3 := #_w1 AND "ST10_SysInput".HMI_Button.ResetButton;
   #_w4 := #_w3 AND NOT #P[6];   // rising edge
   #P[6] := #_w3;
   IF #_w4 THEN "ServoV90_A3".IO.ioManEnale := TRUE; END_IF;
   IF "AlwaysTRUE" THEN
       "ServoV90_A3".In.iManVelocity := "DB_PARAMETERS_TEACH".HMI_PAGE_CONTROL.Speeds.Glue_rotation;
       "ServoV90_A3".In.iManListVelocity := "ServoV90_A3".In.iManVelocity;
   END_IF;
END_REGION

REGION Network 29 (SCL): 382A1 RecipePosition
    IF "Station_Sys".Status.Run THEN
        "ServoV90_A3".Manual.Pos[1].Pos := "ServoV90_A3".Auto.Pos[1].Pos := REAL_TO_DINT("Parameter".AxisRun.Axis[3].Pos1.Position*1000);
        "ServoV90_A3".Manual.Pos[1].Vel := "ServoV90_A3".Auto.Pos[1].Vel := "Parameter".AxisRun.Axis[3].Pos1.Speed;

        "ServoV90_A3".Manual.Pos[2].Pos := "ServoV90_A3".Auto.Pos[2].Pos := REAL_TO_DINT("Parameter".AxisRun.Axis[3].Pos2.Position*1000);
        "ServoV90_A3".Manual.Pos[2].Vel := "ServoV90_A3".Auto.Pos[2].Vel := "Parameter".AxisRun.Axis[3].Pos2.Speed;

        "ServoV90_A3".Manual.Pos[3].Pos := "ServoV90_A3".Auto.Pos[3].Pos := REAL_TO_DINT("Parameter".AxisRun.Axis[3].Pos3.Position*1000);
        "ServoV90_A3".Manual.Pos[3].Vel := "ServoV90_A3".Auto.Pos[3].Vel := "Parameter".AxisRun.Axis[3].Pos3.Speed;

        "ServoV90_A3".Manual.Pos[4].Pos := "ServoV90_A3".Auto.Pos[4].Pos := REAL_TO_DINT("Parameter".AxisRun.Axis[3].Pos4.Position*1000);
        "ServoV90_A3".Manual.Pos[4].Vel := "ServoV90_A3".Auto.Pos[4].Vel := "Parameter".AxisRun.Axis[3].Pos4.Speed;

        "ServoV90_A3".Manual.Pos[5].Pos := "ServoV90_A3".Auto.Pos[5].Pos := REAL_TO_DINT("Parameter".AxisRun.Axis[3].Pos5.Position*1000);
        "ServoV90_A3".Manual.Pos[5].Vel := "ServoV90_A3".Auto.Pos[5].Vel := "Parameter".AxisRun.Axis[3].Pos5.Speed;

        "ServoV90_A3".Manual.Pos[6].Pos := "ServoV90_A3".Auto.Pos[6].Pos := REAL_TO_DINT("Parameter".AxisRun.Axis[3].Pos6.Position*1000);
        "ServoV90_A3".Manual.Pos[6].Vel := "ServoV90_A3".Auto.Pos[6].Vel := "Parameter".AxisRun.Axis[3].Pos6.Speed;

        "ServoV90_A3".Manual.Pos[7].Pos := "ServoV90_A3".Auto.Pos[7].Pos := REAL_TO_DINT("Parameter".AxisRun.Axis[3].Pos7.Position*1000);
        "ServoV90_A3".Manual.Pos[7].Vel := "ServoV90_A3".Auto.Pos[7].Vel := "Parameter".AxisRun.Axis[3].Pos7.Speed;

        "ServoV90_A3".Manual.Pos[8].Pos := "ServoV90_A3".Auto.Pos[8].Pos := REAL_TO_DINT("Parameter".AxisRun.Axis[3].Pos8.Position*1000);
        "ServoV90_A3".Manual.Pos[8].Vel := "ServoV90_A3".Auto.Pos[8].Vel := "Parameter".AxisRun.Axis[3].Pos8.Speed;

        "ServoV90_A3".Manual.Pos[9].Pos := "ServoV90_A3".Auto.Pos[9].Pos := REAL_TO_DINT("Parameter".AxisRun.Axis[3].Pos9.Position*1000);
        "ServoV90_A3".Manual.Pos[9].Vel := "ServoV90_A3".Auto.Pos[9].Vel := "Parameter".AxisRun.Axis[3].Pos9.Speed;

        "ServoV90_A3".Manual.Pos[10].Pos := "ServoV90_A3".Auto.Pos[10].Pos := REAL_TO_DINT("Parameter".AxisRun.Axis[3].Pos10.Position*1000);
        "ServoV90_A3".Manual.Pos[10].Vel := "ServoV90_A3".Auto.Pos[10].Vel := "Parameter".AxisRun.Axis[3].Pos10.Speed;
   END_IF;
END_REGION

REGION Network 30: 382A1 FB
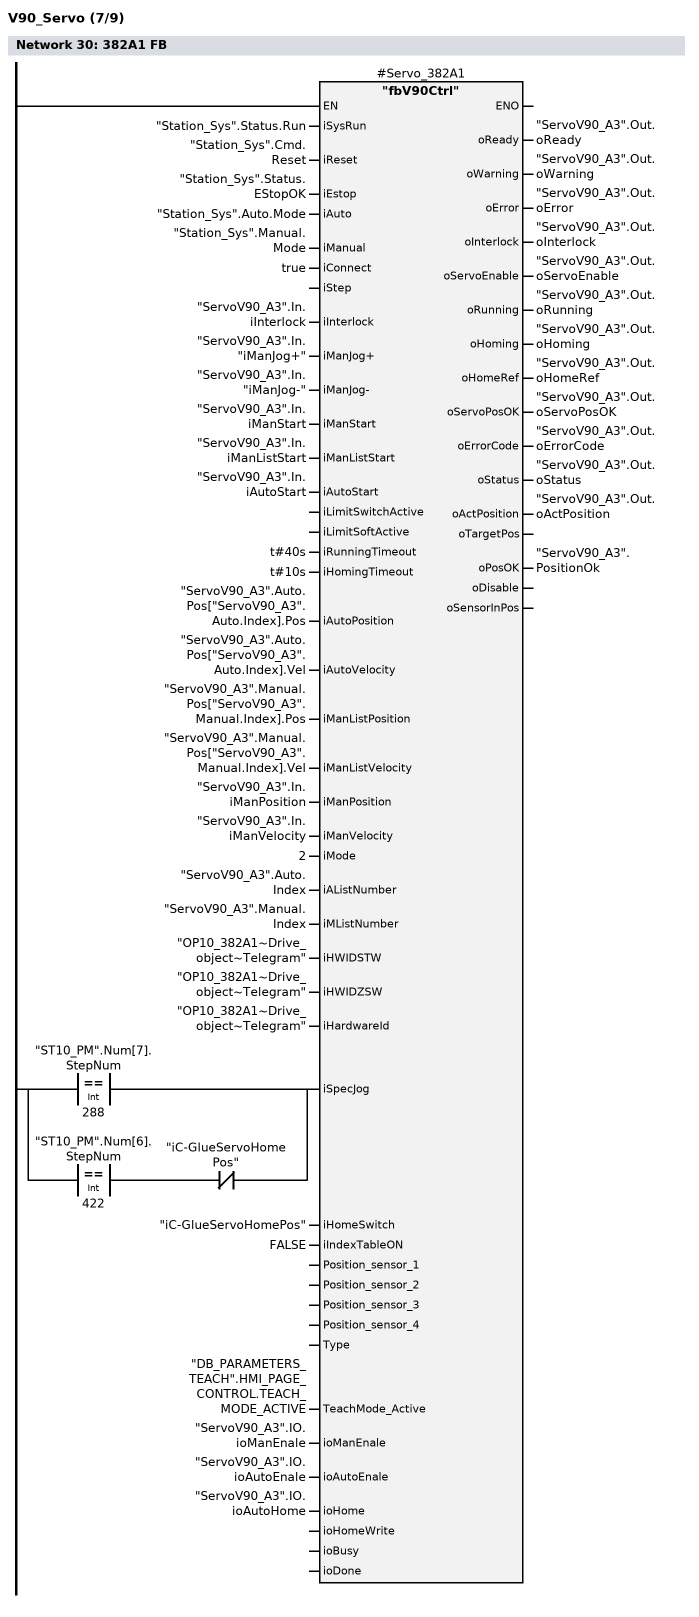
   RUNG wire#powerrail
      #Servo_382A1(iSpecJog := wire#w1, iSysRun := "Station_Sys".Status.Run, iReset := "Station_Sys".Cmd.Reset, iEstop := "Station_Sys".Status.EStopOK, iAuto := "Station_Sys".Auto.Mode, iManual := "Station_Sys".Manual.Mode, iConnect := true, iStep :=, iInterlock := "ServoV90_A3".In.iInterlock, "iManJog+" := "ServoV90_A3".In."iManJog+", "iManJog-" := "ServoV90_A3".In."iManJog-", iManStart := "ServoV90_A3".In.iManStart, iManListStart := "ServoV90_A3".In.iManListStart, iAutoStart := "ServoV90_A3".In.iAutoStart, iLimitSwitchActive :=, iLimitSoftActive :=, iRunningTimeout := t#40s, iHomingTimeout := t#10s, iAutoPosition := "ServoV90_A3".Auto.Pos["ServoV90_A3".Auto.Index].Pos, iAutoVelocity := "ServoV90_A3".Auto.Pos["ServoV90_A3".Auto.Index].Vel, iManListPosition := "ServoV90_A3".Manual.Pos["ServoV90_A3".Manual.Index].Pos, iManListVelocity := "ServoV90_A3".Manual.Pos["ServoV90_A3".Manual.Index].Vel, iManPosition := "ServoV90_A3".In.iManPosition, iManVelocity := "ServoV90_A3".In.iManVelocity, iMode := 2, iAListNumber := "ServoV90_A3".Auto.Index, iMListNumber := "ServoV90_A3".Manual.Index, iHWIDSTW := "OP10_382A1~Drive_object~Telegram", iHWIDZSW := "OP10_382A1~Drive_object~Telegram", iHardwareId := "OP10_382A1~Drive_object~Telegram", iHomeSwitch := "iC-GlueServoHomePos", iIndexTableON := FALSE, Position_sensor_1 :=, Position_sensor_2 :=, Position_sensor_3 :=, Position_sensor_4 :=, "Type" :=, TeachMode_Active := "DB_PARAMETERS_TEACH".HMI_PAGE_CONTROL.TEACH_MODE_ACTIVE, ioManEnale := "ServoV90_A3".IO.ioManEnale, ioAutoEnale := "ServoV90_A3".IO.ioAutoEnale, ioHome := "ServoV90_A3".IO.ioAutoHome, ioHomeWrite :=, ioBusy :=, ioDone :=, oReady => "ServoV90_A3".Out.oReady, oWarning => "ServoV90_A3".Out.oWarning, oError => "ServoV90_A3".Out.oError, oInterlock => "ServoV90_A3".Out.oInterlock, oServoEnable => "ServoV90_A3".Out.oServoEnable, oRunning => "ServoV90_A3".Out.oRunning, oHoming => "ServoV90_A3".Out.oHoming, oHomeRef => "ServoV90_A3".Out.oHomeRef, oServoPosOK => "ServoV90_A3".Out.oServoPosOK, oErrorCode => "ServoV90_A3".Out.oErrorCode, oStatus => "ServoV90_A3".Out.oStatus, oActPosition => "ServoV90_A3".Out.oActPosition, oTargetPos =>, oPosOK => "ServoV90_A3".PositionOk, oDisable =>, oSensorInPos =>)
   END_RUNG
   RUNG wire#powerrail
      { S7_Templates := "SrcType := Int" } EQ_Contact(in1 := "ST10_PM".Num[7].StepNum, in2 := 288)
   END_RUNG wire#w1
   RUNG wire#powerrail
      { S7_Templates := "SrcType := Int" } EQ_Contact(in1 := "ST10_PM".Num[6].StepNum, in2 := 422)
      I_Contact( "iC-GlueServoHomePos" )
   END_RUNG wire#w1
   // the same network as SCL:
   #Servo_382A1(iSysRun := "Station_Sys".Status.Run,   // "fbV90Ctrl"
                iReset := "Station_Sys".Cmd.Reset,
                iEstop := "Station_Sys".Status.EStopOK,
                iAuto := "Station_Sys".Auto.Mode,
                iManual := "Station_Sys".Manual.Mode,
                iConnect := true,
                iInterlock := "ServoV90_A3".In.iInterlock,
                "iManJog+" := "ServoV90_A3".In."iManJog+",
                "iManJog-" := "ServoV90_A3".In."iManJog-",
                iManStart := "ServoV90_A3".In.iManStart,
                iManListStart := "ServoV90_A3".In.iManListStart,
                iAutoStart := "ServoV90_A3".In.iAutoStart,
                iRunningTimeout := t#40s,
                iHomingTimeout := t#10s,
                iAutoPosition := "ServoV90_A3".Auto.Pos["ServoV90_A3".Auto.Index].Pos,
                iAutoVelocity := "ServoV90_A3".Auto.Pos["ServoV90_A3".Auto.Index].Vel,
                iManListPosition := "ServoV90_A3".Manual.Pos["ServoV90_A3".Manual.Index].Pos,
                iManListVelocity := "ServoV90_A3".Manual.Pos["ServoV90_A3".Manual.Index].Vel,
                iManPosition := "ServoV90_A3".In.iManPosition,
                iManVelocity := "ServoV90_A3".In.iManVelocity,
                iMode := 2,
                iAListNumber := "ServoV90_A3".Auto.Index,
                iMListNumber := "ServoV90_A3".Manual.Index,
                iHWIDSTW := "OP10_382A1~Drive_object~Telegram",
                iHWIDZSW := "OP10_382A1~Drive_object~Telegram",
                iHardwareId := "OP10_382A1~Drive_object~Telegram",
                iSpecJog := ("ST10_PM".Num[7].StepNum = 288) OR (("ST10_PM".Num[6].StepNum = 422) AND NOT "iC-GlueServoHomePos"),
                iHomeSwitch := "iC-GlueServoHomePos",
                iIndexTableON := FALSE,
                TeachMode_Active := "DB_PARAMETERS_TEACH".HMI_PAGE_CONTROL.TEACH_MODE_ACTIVE,
                ioManEnale := "ServoV90_A3".IO.ioManEnale,
                ioAutoEnale := "ServoV90_A3".IO.ioAutoEnale,
                ioHome := "ServoV90_A3".IO.ioAutoHome,
                oReady => "ServoV90_A3".Out.oReady,
                oWarning => "ServoV90_A3".Out.oWarning,
                oError => "ServoV90_A3".Out.oError,
                oInterlock => "ServoV90_A3".Out.oInterlock,
                oServoEnable => "ServoV90_A3".Out.oServoEnable,
                oRunning => "ServoV90_A3".Out.oRunning,
                oHoming => "ServoV90_A3".Out.oHoming,
                oHomeRef => "ServoV90_A3".Out.oHomeRef,
                oServoPosOK => "ServoV90_A3".Out.oServoPosOK,
                oErrorCode => "ServoV90_A3".Out.oErrorCode,
                oStatus => "ServoV90_A3".Out.oStatus,
                oActPosition => "ServoV90_A3".Out.oActPosition,
                oPosOK => "ServoV90_A3".PositionOk);
END_REGION

REGION Network 31: 复位启动
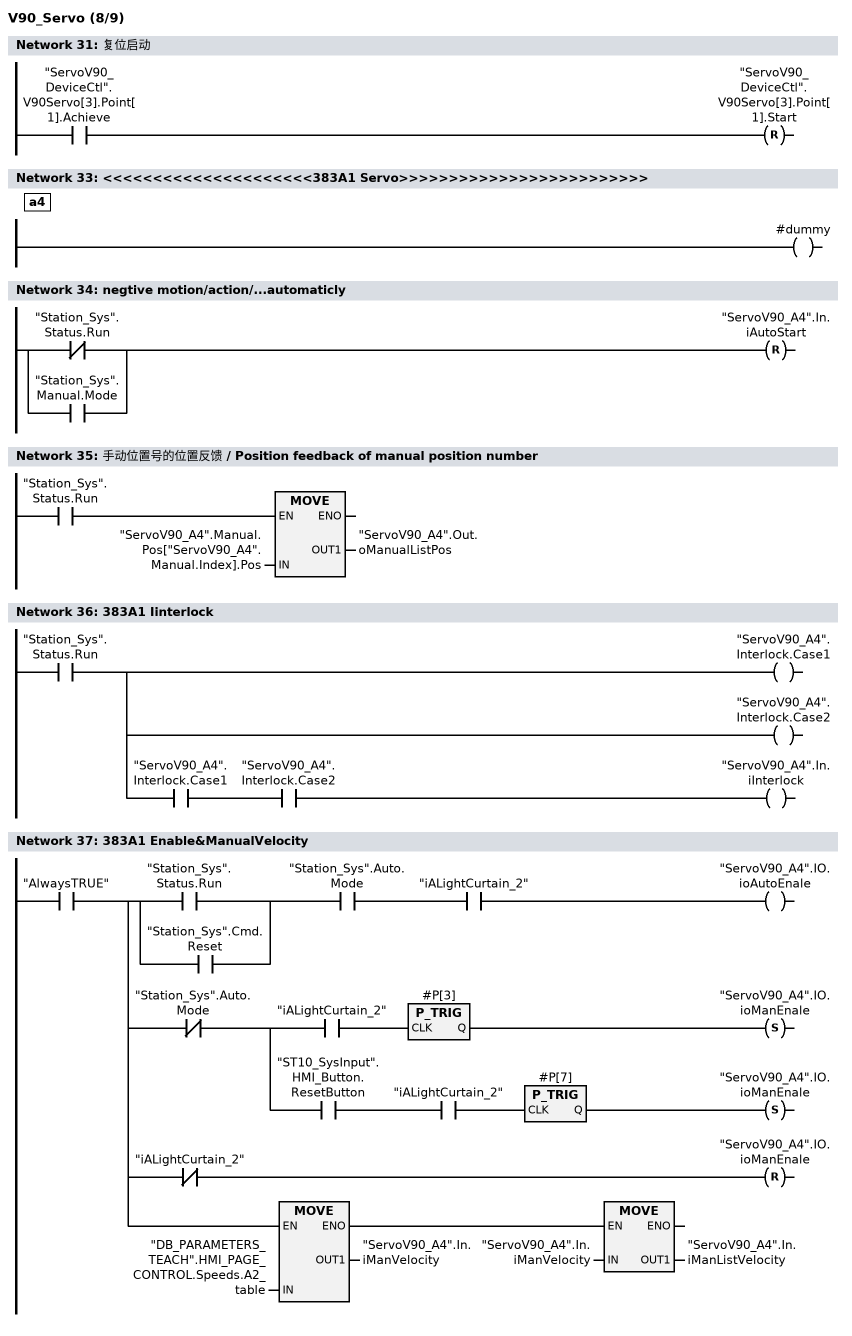
   RUNG wire#powerrail
      Contact( "ServoV90_DeviceCtl".V90Servo[3].Point[1].Achieve )
      R_Coil( "ServoV90_DeviceCtl".V90Servo[3].Point[1].Start )
   END_RUNG
   // the same network as SCL:
   IF "ServoV90_DeviceCtl".V90Servo[3].Point[1].Achieve THEN
       "ServoV90_DeviceCtl".V90Servo[3].Point[1].Start := FALSE;
   END_IF;
END_REGION

REGION Network 32 (SCL): 故障显示 / Fault indication
   //"ST70_DeviceError".Servo2.ServoDriverError := "ServoV90_A3".Out.oError;
END_REGION

REGION Network 33: <<<<<<<<<<<<<<<<<<<<<383A1 Servo>>>>>>>>>>>>>>>>>>>>>>>>>
   Label( a4 )
   RUNG wire#powerrail
      Coil( #dummy )
   END_RUNG
   // the same network as SCL:
   a4:
   #dummy := TRUE;
END_REGION

REGION Network 34: negtive motion/action/...automaticly
   RUNG wire#powerrail
      I_Contact( "Station_Sys".Status.Run )
      wire#w1
      R_Coil( "ServoV90_A4".In.iAutoStart )
   END_RUNG
   RUNG wire#powerrail
      Contact( "Station_Sys".Manual.Mode )
   END_RUNG wire#w1
   // the same network as SCL:
   IF NOT "Station_Sys".Status.Run OR "Station_Sys".Manual.Mode THEN
       "ServoV90_A4".In.iAutoStart := FALSE;
   END_IF;
END_REGION

REGION Network 35: 手动位置号的位置反馈 / Position feedback of manual position number
   RUNG wire#powerrail
      Contact( "Station_Sys".Status.Run )
      Move(in := "ServoV90_A4".Manual.Pos["ServoV90_A4".Manual.Index].Pos, out1 => "ServoV90_A4".Out.oManualListPos)
   END_RUNG
   // the same network as SCL:
   IF "Station_Sys".Status.Run THEN
       "ServoV90_A4".Out.oManualListPos := "ServoV90_A4".Manual.Pos["ServoV90_A4".Manual.Index].Pos;
   END_IF;
END_REGION

REGION Network 36: 383A1 Iinterlock
   RUNG wire#powerrail
      Contact( "Station_Sys".Status.Run )
      wire#w1
      Coil( "ServoV90_A4".Interlock.Case1 )
   END_RUNG
   RUNG wire#w1
      Coil( "ServoV90_A4".Interlock.Case2 )
   END_RUNG
   RUNG wire#w1
      Contact( "ServoV90_A4".Interlock.Case1 )
      Contact( "ServoV90_A4".Interlock.Case2 )
      Coil( "ServoV90_A4".In.iInterlock )
   END_RUNG
   // the same network as SCL:
   "ServoV90_A4".Interlock.Case1 := "Station_Sys".Status.Run;
   "ServoV90_A4".Interlock.Case2 := "Station_Sys".Status.Run;
   "ServoV90_A4".In.iInterlock := "Station_Sys".Status.Run AND "ServoV90_A4".Interlock.Case1 AND "ServoV90_A4".Interlock.Case2;
END_REGION

REGION Network 37: 383A1 Enable&ManualVelocity
   RUNG wire#powerrail
      Contact( "AlwaysTRUE" )
      wire#w1
      Contact( "Station_Sys".Status.Run )
      wire#w2
      Contact( "Station_Sys".Auto.Mode )
      Contact( "iALightCurtain_2" )
      Coil( "ServoV90_A4".IO.ioAutoEnale )
   END_RUNG
   RUNG wire#w1
      Contact( "Station_Sys".Cmd.Reset )
   END_RUNG wire#w2
   RUNG wire#w1
      I_Contact( "Station_Sys".Auto.Mode )
      wire#w3
      Contact( "iALightCurtain_2" )
      P_Trig( #P[3] )
      S_Coil( "ServoV90_A4".IO.ioManEnale )
   END_RUNG
   RUNG wire#w3
      Contact( "ST10_SysInput".HMI_Button.ResetButton )
      Contact( "iALightCurtain_2" )
      P_Trig( #P[7] )
      S_Coil( "ServoV90_A4".IO.ioManEnale )
   END_RUNG
   RUNG wire#w1
      I_Contact( "iALightCurtain_2" )
      R_Coil( "ServoV90_A4".IO.ioManEnale )
   END_RUNG
   RUNG wire#w1
      Move(in := "DB_PARAMETERS_TEACH".HMI_PAGE_CONTROL.Speeds.A2_table, out1 => "ServoV90_A4".In.iManVelocity)
      Move(in := "ServoV90_A4".In.iManVelocity, out1 => "ServoV90_A4".In.iManListVelocity)
   END_RUNG
   // the same network as SCL:
   "ServoV90_A4".IO.ioAutoEnale := "AlwaysTRUE" AND ("Station_Sys".Status.Run OR "Station_Sys".Cmd.Reset) AND "Station_Sys".Auto.Mode AND "iALightCurtain_2";
   #_w1 := "AlwaysTRUE" AND NOT "Station_Sys".Auto.Mode;
   #_w2 := #_w1 AND "iALightCurtain_2";
   #_w3 := #_w2 AND NOT #P[3];   // rising edge
   #P[3] := #_w2;
   IF #_w3 THEN "ServoV90_A4".IO.ioManEnale := TRUE; END_IF;
   #_w4 := #_w1 AND "ST10_SysInput".HMI_Button.ResetButton AND "iALightCurtain_2";
   #_w5 := #_w4 AND NOT #P[7];   // rising edge
   #P[7] := #_w4;
   IF #_w5 THEN "ServoV90_A4".IO.ioManEnale := TRUE; END_IF;
   IF "AlwaysTRUE" AND NOT "iALightCurtain_2" THEN "ServoV90_A4".IO.ioManEnale := FALSE; END_IF;
   IF "AlwaysTRUE" THEN
       "ServoV90_A4".In.iManVelocity := "DB_PARAMETERS_TEACH".HMI_PAGE_CONTROL.Speeds.A2_table;
       "ServoV90_A4".In.iManListVelocity := "ServoV90_A4".In.iManVelocity;
   END_IF;
END_REGION

REGION Network 38 (SCL): 383A1 RecipePosition
   IF "Station_Sys".Status.Run THEN
       "ServoV90_A4".Manual.Pos[1].Pos := "ServoV90_A4".Auto.Pos[1].Pos := REAL_TO_DINT("Parameter".AxisRun.Axis[4].Pos1.Position*1000);
       "ServoV90_A4".Manual.Pos[1].Vel := "ServoV90_A4".Auto.Pos[1].Vel := "Parameter".AxisRun.Axis[4].Pos1.Speed;

       "ServoV90_A4".Manual.Pos[2].Pos := "ServoV90_A4".Auto.Pos[2].Pos := REAL_TO_DINT("Parameter".AxisRun.Axis[4].Pos2.Position*1000);
       "ServoV90_A4".Manual.Pos[2].Vel := "ServoV90_A4".Auto.Pos[2].Vel := "Parameter".AxisRun.Axis[4].Pos2.Speed;

       "ServoV90_A4".Manual.Pos[3].Pos := "ServoV90_A4".Auto.Pos[3].Pos := REAL_TO_DINT("Parameter".AxisRun.Axis[4].Pos3.Position*1000);
       "ServoV90_A4".Manual.Pos[3].Vel := "ServoV90_A4".Auto.Pos[3].Vel := "Parameter".AxisRun.Axis[4].Pos3.Speed;

       "ServoV90_A4".Manual.Pos[4].Pos := "ServoV90_A4".Auto.Pos[4].Pos := REAL_TO_DINT("Parameter".AxisRun.Axis[4].Pos4.Position*1000);
       "ServoV90_A4".Manual.Pos[4].Vel := "ServoV90_A4".Auto.Pos[4].Vel := "Parameter".AxisRun.Axis[4].Pos4.Speed;

       "ServoV90_A4".Manual.Pos[5].Pos := "ServoV90_A4".Auto.Pos[5].Pos := REAL_TO_DINT("Parameter".AxisRun.Axis[4].Pos5.Position*1000);
       "ServoV90_A4".Manual.Pos[5].Vel := "ServoV90_A4".Auto.Pos[5].Vel := "Parameter".AxisRun.Axis[4].Pos5.Speed;

       "ServoV90_A4".Manual.Pos[6].Pos := "ServoV90_A4".Auto.Pos[6].Pos := REAL_TO_DINT("Parameter".AxisRun.Axis[4].Pos6.Position*1000);
       "ServoV90_A4".Manual.Pos[6].Vel := "ServoV90_A4".Auto.Pos[6].Vel := "Parameter".AxisRun.Axis[4].Pos6.Speed;

       "ServoV90_A4".Manual.Pos[7].Pos := "ServoV90_A4".Auto.Pos[7].Pos := REAL_TO_DINT("Parameter".AxisRun.Axis[4].Pos7.Position*1000);
       "ServoV90_A4".Manual.Pos[7].Vel := "ServoV90_A4".Auto.Pos[7].Vel := "Parameter".AxisRun.Axis[4].Pos7.Speed;

       "ServoV90_A4".Manual.Pos[8].Pos := "ServoV90_A4".Auto.Pos[8].Pos := REAL_TO_DINT("Parameter".AxisRun.Axis[4].Pos8.Position*1000);
       "ServoV90_A4".Manual.Pos[8].Vel := "ServoV90_A4".Auto.Pos[8].Vel := "Parameter".AxisRun.Axis[4].Pos8.Speed;

       "ServoV90_A4".Manual.Pos[9].Pos := "ServoV90_A4".Auto.Pos[9].Pos := REAL_TO_DINT("Parameter".AxisRun.Axis[4].Pos9.Position*1000);
       "ServoV90_A4".Manual.Pos[9].Vel := "ServoV90_A4".Auto.Pos[9].Vel := "Parameter".AxisRun.Axis[4].Pos9.Speed;

       "ServoV90_A4".Manual.Pos[10].Pos := "ServoV90_A4".Auto.Pos[10].Pos := REAL_TO_DINT("Parameter".AxisRun.Axis[4].Pos10.Position*1000);
       "ServoV90_A4".Manual.Pos[10].Vel := "ServoV90_A4".Auto.Pos[10].Vel := "Parameter".AxisRun.Axis[4].Pos10.Speed;
   END_IF;
END_REGION

REGION Network 39: 383A1 FB
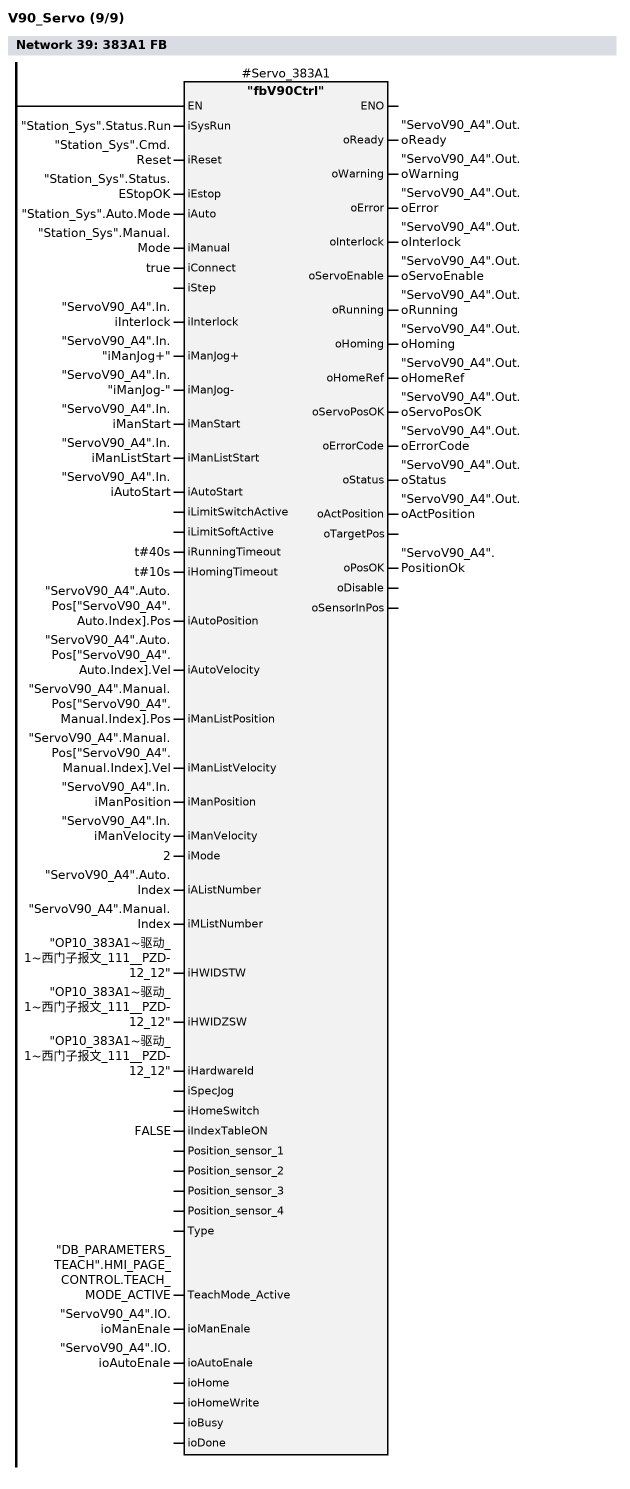
   RUNG wire#powerrail
      #Servo_383A1(iSysRun := "Station_Sys".Status.Run, iReset := "Station_Sys".Cmd.Reset, iEstop := "Station_Sys".Status.EStopOK, iAuto := "Station_Sys".Auto.Mode, iManual := "Station_Sys".Manual.Mode, iConnect := true, iStep :=, iInterlock := "ServoV90_A4".In.iInterlock, "iManJog+" := "ServoV90_A4".In."iManJog+", "iManJog-" := "ServoV90_A4".In."iManJog-", iManStart := "ServoV90_A4".In.iManStart, iManListStart := "ServoV90_A4".In.iManListStart, iAutoStart := "ServoV90_A4".In.iAutoStart, iLimitSwitchActive :=, iLimitSoftActive :=, iRunningTimeout := t#40s, iHomingTimeout := t#10s, iAutoPosition := "ServoV90_A4".Auto.Pos["ServoV90_A4".Auto.Index].Pos, iAutoVelocity := "ServoV90_A4".Auto.Pos["ServoV90_A4".Auto.Index].Vel, iManListPosition := "ServoV90_A4".Manual.Pos["ServoV90_A4".Manual.Index].Pos, iManListVelocity := "ServoV90_A4".Manual.Pos["ServoV90_A4".Manual.Index].Vel, iManPosition := "ServoV90_A4".In.iManPosition, iManVelocity := "ServoV90_A4".In.iManVelocity, iMode := 2, iAListNumber := "ServoV90_A4".Auto.Index, iMListNumber := "ServoV90_A4".Manual.Index, iHWIDSTW := "OP10_383A1~驱动_1~西门子报文_111__PZD-12_12", iHWIDZSW := "OP10_383A1~驱动_1~西门子报文_111__PZD-12_12", iHardwareId := "OP10_383A1~驱动_1~西门子报文_111__PZD-12_12", iSpecJog :=, iHomeSwitch :=, iIndexTableON := FALSE, Position_sensor_1 :=, Position_sensor_2 :=, Position_sensor_3 :=, Position_sensor_4 :=, "Type" :=, TeachMode_Active := "DB_PARAMETERS_TEACH".HMI_PAGE_CONTROL.TEACH_MODE_ACTIVE, ioManEnale := "ServoV90_A4".IO.ioManEnale, ioAutoEnale := "ServoV90_A4".IO.ioAutoEnale, ioHome :=, ioHomeWrite :=, ioBusy :=, ioDone :=, oReady => "ServoV90_A4".Out.oReady, oWarning => "ServoV90_A4".Out.oWarning, oError => "ServoV90_A4".Out.oError, oInterlock => "ServoV90_A4".Out.oInterlock, oServoEnable => "ServoV90_A4".Out.oServoEnable, oRunning => "ServoV90_A4".Out.oRunning, oHoming => "ServoV90_A4".Out.oHoming, oHomeRef => "ServoV90_A4".Out.oHomeRef, oServoPosOK => "ServoV90_A4".Out.oServoPosOK, oErrorCode => "ServoV90_A4".Out.oErrorCode, oStatus => "ServoV90_A4".Out.oStatus, oActPosition => "ServoV90_A4".Out.oActPosition, oTargetPos =>, oPosOK => "ServoV90_A4".PositionOk, oDisable =>, oSensorInPos =>)
   END_RUNG
   // the same network as SCL:
   #Servo_383A1(iSysRun := "Station_Sys".Status.Run,   // "fbV90Ctrl"
                iReset := "Station_Sys".Cmd.Reset,
                iEstop := "Station_Sys".Status.EStopOK,
                iAuto := "Station_Sys".Auto.Mode,
                iManual := "Station_Sys".Manual.Mode,
                iConnect := true,
                iInterlock := "ServoV90_A4".In.iInterlock,
                "iManJog+" := "ServoV90_A4".In."iManJog+",
                "iManJog-" := "ServoV90_A4".In."iManJog-",
                iManStart := "ServoV90_A4".In.iManStart,
                iManListStart := "ServoV90_A4".In.iManListStart,
                iAutoStart := "ServoV90_A4".In.iAutoStart,
                iRunningTimeout := t#40s,
                iHomingTimeout := t#10s,
                iAutoPosition := "ServoV90_A4".Auto.Pos["ServoV90_A4".Auto.Index].Pos,
                iAutoVelocity := "ServoV90_A4".Auto.Pos["ServoV90_A4".Auto.Index].Vel,
                iManListPosition := "ServoV90_A4".Manual.Pos["ServoV90_A4".Manual.Index].Pos,
                iManListVelocity := "ServoV90_A4".Manual.Pos["ServoV90_A4".Manual.Index].Vel,
                iManPosition := "ServoV90_A4".In.iManPosition,
                iManVelocity := "ServoV90_A4".In.iManVelocity,
                iMode := 2,
                iAListNumber := "ServoV90_A4".Auto.Index,
                iMListNumber := "ServoV90_A4".Manual.Index,
                iHWIDSTW := "OP10_383A1~驱动_1~西门子报文_111__PZD-12_12",
                iHWIDZSW := "OP10_383A1~驱动_1~西门子报文_111__PZD-12_12",
                iHardwareId := "OP10_383A1~驱动_1~西门子报文_111__PZD-12_12",
                iIndexTableON := FALSE,
                TeachMode_Active := "DB_PARAMETERS_TEACH".HMI_PAGE_CONTROL.TEACH_MODE_ACTIVE,
                ioManEnale := "ServoV90_A4".IO.ioManEnale,
                ioAutoEnale := "ServoV90_A4".IO.ioAutoEnale,
                oReady => "ServoV90_A4".Out.oReady,
                oWarning => "ServoV90_A4".Out.oWarning,
                oError => "ServoV90_A4".Out.oError,
                oInterlock => "ServoV90_A4".Out.oInterlock,
                oServoEnable => "ServoV90_A4".Out.oServoEnable,
                oRunning => "ServoV90_A4".Out.oRunning,
                oHoming => "ServoV90_A4".Out.oHoming,
                oHomeRef => "ServoV90_A4".Out.oHomeRef,
                oServoPosOK => "ServoV90_A4".Out.oServoPosOK,
                oErrorCode => "ServoV90_A4".Out.oErrorCode,
                oStatus => "ServoV90_A4".Out.oStatus,
                oActPosition => "ServoV90_A4".Out.oActPosition,
                oPosOK => "ServoV90_A4".PositionOk);
END_REGION

REGION Network 40 (SCL): 故障显示 / Fault indication
   //"ST70_DeviceError".Servo2.ServoDriverError := "ServoV90_A4".Out.oError;
END_REGION

REGION Network 41: *********************************伺服位置判断**********************************************
END_REGION

REGION Network 42 (SCL): 伺服位置判断 / Servo position judgment
   FOR "ServoV90_DeviceCtl".V90Servo[1].i := 1 TO 12 BY 1 DO
       "ServoV90_DeviceCtl".V90Servo[1].Pos.List["ServoV90_DeviceCtl".V90Servo[1].i].Pos := "ServoV90_A1".Auto.Pos["ServoV90_DeviceCtl".V90Servo[1].i].Pos;
       "ServoV90_DeviceCtl".V90Servo[1].Pos.List["ServoV90_DeviceCtl".V90Servo[1].i].Vel := "ServoV90_A1".Auto.Pos["ServoV90_DeviceCtl".V90Servo[1].i].Vel;

       "ServoV90_DeviceCtl".V90Servo[2].Pos.List["ServoV90_DeviceCtl".V90Servo[1].i].Pos := "ServoV90_A2".Auto.Pos["ServoV90_DeviceCtl".V90Servo[1].i].Pos;
       "ServoV90_DeviceCtl".V90Servo[2].Pos.List["ServoV90_DeviceCtl".V90Servo[1].i].Vel := "ServoV90_A2".Auto.Pos["ServoV90_DeviceCtl".V90Servo[1].i].Vel;

       "ServoV90_DeviceCtl".V90Servo[3].Pos.List["ServoV90_DeviceCtl".V90Servo[1].i].Pos := "ServoV90_A3".Auto.Pos["ServoV90_DeviceCtl".V90Servo[1].i].Pos;
       "ServoV90_DeviceCtl".V90Servo[3].Pos.List["ServoV90_DeviceCtl".V90Servo[1].i].Vel := "ServoV90_A3".Auto.Pos["ServoV90_DeviceCtl".V90Servo[1].i].Vel;

       "ServoV90_DeviceCtl".V90Servo[4].Pos.List["ServoV90_DeviceCtl".V90Servo[1].i].Pos := "ServoV90_A4".Auto.Pos["ServoV90_DeviceCtl".V90Servo[1].i].Pos;
       "ServoV90_DeviceCtl".V90Servo[4].Pos.List["ServoV90_DeviceCtl".V90Servo[1].i].Vel := "ServoV90_A4".Auto.Pos["ServoV90_DeviceCtl".V90Servo[1].i].Vel;

   END_FOR;

   (******************************************************* SV1 ********************************************************************)   
   //伺服位置判断
   #"Servo1"(iRef_Homed :=   "ServoV90_A1".Out.oHomeRef,
                             iStandstill := FALSE,
                             iReset := "Station_Sys".Cmd.Reset,
                             interlcok:="ServoV90_A1".In.iInterlock,
                             "iActual Posi" :="ServoV90_A1".Out.oActPosition,
                             "iTol+" := 50,
                             "iTol-" := 50,
                             iStartTon := T#100mS,
                             ioPoint:="ServoV90_DeviceCtl".V90Servo[1].Point,
                             oStartPos => #Sevro1StartList,
                             ioList := "ServoV90_DeviceCtl".V90Servo[1].Pos,
                             ioPosNumberSelect := "ServoV90_DeviceCtl".V90Servo[1].nPositionListNo);

   IF "ServoV90_DeviceCtl".V90Servo[1].nPositionListNo = 0 THEN
      "ServoV90_DeviceCtl".V90Servo[1].nPositionListNo:= 1 ;
   END_IF;

    //伺服位置号给定
                   // IF NOT "D-2 ModuleD-2 横向抓取移栽/拍照/旋转_IDB".伺服到下料位.X THEN
                   //     "ServoV90_A1".Auto.Index := "ServoV90_DeviceCtl".V90Servo[1].nPositionListNo;
                   // END_IF;

                  "ServoV90_A1".Auto.Index := "ServoV90_DeviceCtl".V90Servo[1].nPositionListNo;

   //伺服启动
                   "ServoV90_A1".In.iAutoStart := #Sevro1StartList;


   (******************************************************* SV2 ********************************************************************)                
   //伺服位置判断
   #"Servo2"(iRef_Homed := "ServoV90_A2".Out.oHomeRef,
             iStandstill := FALSE,
             iReset := "Station_Sys".Cmd.Reset,
             interlcok := "ServoV90_A2".In.iInterlock,
             "iActual Posi" := "ServoV90_A2".Out.oActPosition,
             "iTol+" := 50,
             "iTol-" := 50,
             iStartTon := T#100mS,
             ioPoint := "ServoV90_DeviceCtl".V90Servo[2].Point,
             oStartPos => #Sevro2StartList,
             ioList := "ServoV90_DeviceCtl".V90Servo[2].Pos,
             ioPosNumberSelect := "ServoV90_DeviceCtl".V90Servo[2].nPositionListNo);

   IF "ServoV90_DeviceCtl".V90Servo[2].nPositionListNo = 0 THEN
       "ServoV90_DeviceCtl".V90Servo[2].nPositionListNo := 1;
   END_IF;

   //伺服位置号给定
   // IF NOT "D-3 ModuleD-3从转台下料到托盘移栽机构_IDB".移栽伺服到取料位1.X THEN
   //     "ServoV90_A2".Auto.Index := "ServoV90_DeviceCtl".CMMTServo[2].nPositionListNo;
   // END_IF;

   "ServoV90_A2".Auto.Index := "ServoV90_DeviceCtl".V90Servo[2].nPositionListNo;

   //伺服启动
   "ServoV90_A2".In.iAutoStart := #Sevro2StartList;


   (******************************************************* SV3 ********************************************************************)
   //伺服位置判断
   #"Servo3"(iRef_Homed := "ServoV90_A3".Out.oHomeRef,
             iStandstill := FALSE,
             iReset := "Station_Sys".Cmd.Reset,
             interlcok := "ServoV90_A3".In.iInterlock,
             "iActual Posi" := "ServoV90_A3".Out.oActPosition,
             "iTol+" := 50,
             "iTol-" := 50,
             iStartTon := T#100mS,
             ioPoint := "ServoV90_DeviceCtl".V90Servo[3].Point,
             oStartPos => #Sevro3StartList,
             ioList := "ServoV90_DeviceCtl".V90Servo[3].Pos,
             ioPosNumberSelect := "ServoV90_DeviceCtl".V90Servo[3].nPositionListNo);

   IF "ServoV90_DeviceCtl".V90Servo[3].nPositionListNo = 0 THEN
       "ServoV90_DeviceCtl".V90Servo[3].nPositionListNo := 1;
   END_IF;
   //伺服位置号给定
   // IF NOT "D-3 ModuleD-3从转台下料到托盘移栽机构_IDB".移栽伺服到取料位1.X THEN
   //     "ServoV90_A2".Auto.Index := "ServoV90_DeviceCtl".V90Servo[2].nPositionListNo;
   // END_IF;

   "ServoV90_A3".Auto.Index := "ServoV90_DeviceCtl".V90Servo[3].nPositionListNo;

   //伺服启动
   "ServoV90_A3".In.iAutoStart := #Sevro3StartList;


   (******************************************************* SV4 ********************************************************************)
   //伺服位置判断
   #"Servo4"(iRef_Homed := "ServoV90_A4".Out.oHomeRef,
             iStandstill := FALSE,
             iReset := "Station_Sys".Cmd.Reset,
             interlcok := "ServoV90_A4".In.iInterlock,
             "iActual Posi" := "ServoV90_A4".Out.oActPosition,
             "iTol+" := 50,
             "iTol-" := 50,
             iStartTon := T#100mS,
             ioPoint := "ServoV90_DeviceCtl".V90Servo[4].Point,
             oStartPos => #Sevro4StartList,
             ioList := "ServoV90_DeviceCtl".V90Servo[4].Pos,
             ioPosNumberSelect := "ServoV90_DeviceCtl".V90Servo[4].nPositionListNo);

   IF "ServoV90_DeviceCtl".V90Servo[4].nPositionListNo = 0 THEN
       "ServoV90_DeviceCtl".V90Servo[4].nPositionListNo := 1;
   END_IF;

   //伺服位置号给定
   // IF NOT "D-3 ModuleD-3从转台下料到托盘移栽机构_IDB".移栽伺服到取料位1.X THEN
   //     "ServoV90_A2".Auto.Index := "ServoV90_DeviceCtl".V90Servo[2].nPositionListNo;
   // END_IF;

   "ServoV90_A4".Auto.Index := "ServoV90_DeviceCtl".V90Servo[4].nPositionListNo;

   //伺服启动
   "ServoV90_A4".In.iAutoStart := #Sevro4StartList;
END_REGION

REGION Network 43 (SCL): 初始化脉冲 置位手动使能 / The initial pulse set function was manually enabled
   IF "FirstScan" THEN
       "ServoV90_A1".IO.ioManEnale := TRUE;
       "ServoV90_A2".IO.ioManEnale := TRUE;
       "ServoV90_A3".IO.ioManEnale := TRUE;
       "ServoV90_A4".IO.ioManEnale := TRUE;
   END_IF;
END_REGION
END_FUNCTION_BLOCK
